	IQ_stMeldung.bMeldFBError_ErrorDiag	:= FALSE;
	IQ_stMeldung.bMeldFBError_ErrorState:= FALSE;
	IQ_stMeldung.sMeldFBError_ErrorDiag	:= '';
	IQ_stMeldung.sMeldFBError_ErrorState:= '';
	
	sFB				:= CONCAT('TwinSAFE Gruppe',INT_TO_STRING(I_nGrpId));
	sFB				:= CONCAT(sFB,' => ');
	sFB				:= CONCAT(sFB,'FB');
	sFB				:= CONCAT(sFB,INT_TO_STRING(I_nFBId));
	sFB				:= CONCAT(sFB,' ');
	sFB				:= CONCAT(sFB,I_sFBName);
	sFB				:= CONCAT(sFB,' => ');

	(* ========================================================= *)
	(* State *)
	CASE I_stInfoData.nMapState OF
		0:	IQ_stMeldung.sMeldFBError_ErrorState	:= 'undefiniert';
			act_State();

		1:	IQ_stMeldung.sMeldFBError_ErrorState	:= 'Run';

		2:	IQ_stMeldung.sMeldFBError_ErrorState	:= 'Stop';

		3:	IQ_stMeldung.sMeldFBError_ErrorState	:= 'Safe';

	ELSE	IQ_stMeldung.sMeldFBError_ErrorState	:= 'Error';
			act_State();
	END_CASE

	(* ========================================================= *)
	(* Diagnose *)
	(*	stInfoData.uiMapDiag	immer gleich 0*)
	CASE I_stInfoData.nMapState OF
		0:	;
	END_CASE

	(* ========================================================= *)
	(*BE*)
END_ACTION

ACTION actInfoConnectionShutDown:
	(* TwinSAFE-Funktionsbaustein FB Connection Shutdown *)
	(* ========================================================= *)

	IQ_stMeldung.bMeldFBError_ErrorDiag	:= FALSE;
	IQ_stMeldung.bMeldFBError_ErrorState:= FALSE;
	IQ_stMeldung.sMeldFBError_ErrorDiag	:= '';
	IQ_stMeldung.sMeldFBError_ErrorState:= '';
	
	sFB				:= CONCAT('TwinSAFE Gruppe',INT_TO_STRING(I_nGrpId));
	sFB				:= CONCAT(sFB,' => ');
	sFB				:= CONCAT(sFB,'FB');
	sFB				:= CONCAT(sFB,INT_TO_STRING(I_nFBId));
	sFB				:= CONCAT(sFB,' ');
	sFB				:= CONCAT(sFB,I_sFBName);
	sFB				:= CONCAT(sFB,' => ');

	(* ========================================================= *)
	(* State *)
	CASE I_stInfoData.nMapState OF
		0:	IQ_stMeldung.sMeldFBError_ErrorState	:= 'undefiniert';
			act_State();

		2:	IQ_stMeldung.sMeldFBError_ErrorState	:= 'Stop';

		3:	IQ_stMeldung.sMeldFBError_ErrorState	:= 'Safe';

		4:	IQ_stMeldung.sMeldFBError_ErrorState	:= 'Error';
			act_State();

		5:	IQ_stMeldung.sMeldFBError_ErrorState	:= 'Reset';

		10:IQ_stMeldung.sMeldFBError_ErrorState	:= 'Active';

		11:IQ_stMeldung.sMeldFBError_ErrorState	:= 'Deactive';

	ELSE	IQ_stMeldung.sMeldFBError_ErrorState	:= 'Error';
			act_State();
	END_CASE

	(* ========================================================= *)
	(* Diagnose *)
	(*	stInfoData.uiMapDiag	immer gleich 0*)
	CASE I_stInfoData.nMapDiag OF
		0: IQ_stMeldung.sMeldFBError_ErrorDiag	 :='-';
	ELSE
		IF I_stInfoData.nMapDiag.0 THEN
			IQ_stMeldung.sMeldFBError_ErrorDiag	:='Diskrepanz Fehler Eingangsgruppe 1 => Safety Input => ';
			IQ_stMeldung.sMeldFBError_ErrorDiag	:= CONCAT(IQ_stMeldung.sMeldFBError_ErrorDiag,I_sNameEinGruppe1);
			act_Diag();
		END_IF
	END_CASE

	(* ========================================================= *)
	(*BE*)
END_ACTION

ACTION actInfoDecoupler:
	(* TwinSAFE-Funktionsbaustein FB Decouple*)
	(* ========================================================= *)

	IQ_stMeldung.bMeldFBError_ErrorDiag	:= FALSE;
	IQ_stMeldung.bMeldFBError_ErrorState:= FALSE;
	IQ_stMeldung.sMeldFBError_ErrorDiag	:= '';
	IQ_stMeldung.sMeldFBError_ErrorState:= '';
	
	sFB				:= CONCAT('TwinSAFE Gruppe',INT_TO_STRING(I_nGrpId));
	sFB				:= CONCAT(sFB,' => ');
	sFB				:= CONCAT(sFB,'FB');
	sFB				:= CONCAT(sFB,INT_TO_STRING(I_nFBId));
	sFB				:= CONCAT(sFB,' ');
	sFB				:= CONCAT(sFB,I_sFBName);
	sFB				:= CONCAT(sFB,' => ');

	(* ========================================================= *)
	(* State *)
	CASE I_stInfoData.nMapState OF
		0:	IQ_stMeldung.sMeldFBError_ErrorState	:= 'undefiniert';
			act_State();

		1:	IQ_stMeldung.sMeldFBError_ErrorState	:= 'Run';

		2:	IQ_stMeldung.sMeldFBError_ErrorState	:= 'Stop';

	ELSE	IQ_stMeldung.sMeldFBError_ErrorState	:= 'Error';
			act_State();
	END_CASE

	(* ========================================================= *)
	(* Diagnose *)
	(*	stInfoData.uiMapDiag	immer gleich 0*)
	CASE I_stInfoData.nMapState OF
		0:	;
	END_CASE

	(* ========================================================= *)
	(*BE*)
END_ACTION

ACTION actInfoEDM:
	(* TwinSAFE-Funktionsbaustein FB EDM *)
	(* ========================================================= *)

	IQ_stMeldung.bMeldFBError_ErrorDiag	:= FALSE;
	IQ_stMeldung.bMeldFBError_ErrorState:= FALSE;
	IQ_stMeldung.sMeldFBError_ErrorDiag	:= '';
	IQ_stMeldung.sMeldFBError_ErrorState:= '';

	sFB				:= CONCAT('TwinSAFE Gruppe',INT_TO_STRING(I_nGrpId));
	sFB				:= CONCAT(sFB,' => ');
	sFB				:= CONCAT(sFB,'FB');
	sFB				:= CONCAT(sFB,INT_TO_STRING(I_nFBId));
	sFB				:= CONCAT(sFB,' ');
	sFB				:= CONCAT(sFB,I_sFBName);
	sFB				:= CONCAT(sFB,' => ');

	(* ========================================================= *)
	(* State *)
	CASE I_stInfoData.nMapState OF
		0:	IQ_stMeldung.sMeldFBError_ErrorState	:= 'undefiniert';
			act_State();

		2:	IQ_stMeldung.sMeldFBError_ErrorState	:= 'Stop';

		4:	IQ_stMeldung.sMeldFBError_ErrorState	:= 'Error';
			act_State();

		5:	IQ_stMeldung.sMeldFBError_ErrorState	:= 'Reset';

		14:IQ_stMeldung.sMeldFBError_ErrorState	:= 'MON_OFF';

		15:IQ_stMeldung.sMeldFBError_ErrorState	:= 'MON_ON';

	ELSE	IQ_stMeldung.sMeldFBError_ErrorState	:= 'Error';
			act_State();
	END_CASE

	(* ========================================================= *)
	(* Diagnose *)
	CASE I_stInfoData.nMapDiag OF
		0: ;
	ELSE
		IF I_stInfoData.nMapDiag.0 THEN
			IQ_stMeldung.sMeldFBError_ErrorDiag	:='Switch OFF Timer abgelaufen';
			act_Diag();
		END_IF
		IF I_stInfoData.nMapDiag.1 THEN
			IQ_stMeldung.sMeldFBError_ErrorDiag	:='Switch ON Timer abgelaufen';
			act_Diag();
		END_IF
	END_CASE

	(* ========================================================= *)
	(*BE*)
END_ACTION

ACTION actInfoEStop:
	(* TwinSAFE-Funktionsbaustein FB EStop *)
	(* ========================================================= *)

	IQ_stMeldung.bMeldFBError_ErrorDiag	:= FALSE;
	IQ_stMeldung.bMeldFBError_ErrorState:= FALSE;
	IQ_stMeldung.sMeldFBError_ErrorDiag	:= '';
	IQ_stMeldung.sMeldFBError_ErrorState:= '';

	sFB				:= CONCAT('TwinSAFE Gruppe',INT_TO_STRING(I_nGrpId));
	sFB				:= CONCAT(sFB,' => ');
	sFB				:= CONCAT(sFB,'FB');
	sFB				:= CONCAT(sFB,INT_TO_STRING(I_nFBId));
	sFB				:= CONCAT(sFB,' ');
	sFB				:= CONCAT(sFB,I_sFBName);
	sFB				:= CONCAT(sFB,' => ');
	(* ========================================================= *)
	(* State *)
	CASE I_stInfoData.nMapState OF
		0:	IQ_stMeldung.sMeldFBError_ErrorState	:= 'undefiniert';
			act_State();

		1:	IQ_stMeldung.sMeldFBError_ErrorState	:= 'Run';

		2:	IQ_stMeldung.sMeldFBError_ErrorState	:= 'Stop';

		3:	IQ_stMeldung.sMeldFBError_ErrorState	:= 'Safe';

		4:	IQ_stMeldung.sMeldFBError_ErrorState	:= 'Error';
			act_State();

		5:	IQ_stMeldung.sMeldFBError_ErrorState	:= 'Reset';

		6:	IQ_stMeldung.sMeldFBError_ErrorState	:= 'Start';

		8:	IQ_stMeldung.sMeldFBError_ErrorState	:= 'DelayOut';

	ELSE	IQ_stMeldung.sMeldFBError_ErrorState	:= 'Error';
			act_State();
	END_CASE

	(* ========================================================= *)
	(* Diagnose *)
	CASE I_stInfoData.nMapDiag OF
		0: IQ_stMeldung.sMeldFBError_ErrorDiag :='-';
	ELSE
		IF I_stInfoData.nMapDiag.0 THEN
			IQ_stMeldung.sMeldFBError_ErrorDiag	:='Diskrepanz Fehler Eingangsgruppe 1 => Safety Input => ';
			IQ_stMeldung.sMeldFBError_ErrorDiag	:= CONCAT(IQ_stMeldung.sMeldFBError_ErrorDiag,I_sNameEinGruppe1);
			act_Diag();
		END_IF

		IF I_stInfoData.nMapDiag.1 THEN
			IQ_stMeldung.sMeldFBError_ErrorDiag	:='Diskrepanz Fehler Eingangsgruppe 2 => Safety Input => ';
			IQ_stMeldung.sMeldFBError_ErrorDiag	:= CONCAT(IQ_stMeldung.sMeldFBError_ErrorDiag,I_sNameEinGruppe2);
			act_Diag();
		END_IF

		IF I_stInfoData.nMapDiag.2 THEN
			IQ_stMeldung.sMeldFBError_ErrorDiag	:='Diskrepanz Fehler Eingangsgruppe 3 => Safety Input => ';
			IQ_stMeldung.sMeldFBError_ErrorDiag	:= CONCAT(IQ_stMeldung.sMeldFBError_ErrorDiag,I_sNameEinGruppe3);
			act_Diag();
		END_IF

		IF I_stInfoData.nMapDiag.3 THEN
			IQ_stMeldung.sMeldFBError_ErrorDiag	:='Diskrepanz Fehler Eingangsgruppe 4 => Safety Input => ';
			IQ_stMeldung.sMeldFBError_ErrorDiag	:= CONCAT(IQ_stMeldung.sMeldFBError_ErrorDiag,I_sNameEinGruppe4);
			act_Diag();
		END_IF

		IF I_stInfoData.nMapDiag.4 THEN
			IQ_stMeldung.sMeldFBError_ErrorDiag	:='Rueckfuehrkreis Fehler EDM1 => Safety Input => ';
			IQ_stMeldung.sMeldFBError_ErrorDiag	:= CONCAT(IQ_stMeldung.sMeldFBError_ErrorDiag,I_sNameEMD1);
			act_Diag();
		END_IF

		IF I_stInfoData.nMapDiag.5 THEN
			IQ_stMeldung.sMeldFBError_ErrorDiag	:='Rueckfuehrkreis Fehler EDM2 => Safety Input => ';
			IQ_stMeldung.sMeldFBError_ErrorDiag	:= CONCAT(IQ_stMeldung.sMeldFBError_ErrorDiag,I_sNameEMD2);
			act_Diag();
		END_IF
	END_CASE

	(* ========================================================= *)
	(*BE*)
END_ACTION

ACTION actInfoMON:
	(* TwinSAFE-Funktionsbaustein FB MOM *)
	(* ========================================================= *)

	IQ_stMeldung.bMeldFBError_ErrorDiag	:= FALSE;
	IQ_stMeldung.bMeldFBError_ErrorState:= FALSE;
	IQ_stMeldung.sMeldFBError_ErrorDiag	:= '';
	IQ_stMeldung.sMeldFBError_ErrorState:= '';

	sFB				:= CONCAT('TwinSAFE Gruppe',INT_TO_STRING(I_nGrpId));
	sFB				:= CONCAT(sFB,' => ');
	sFB				:= CONCAT(sFB,'FB');
	sFB				:= CONCAT(sFB,INT_TO_STRING(I_nFBId));
	sFB				:= CONCAT(sFB,' ');
	sFB				:= CONCAT(sFB,I_sFBName);
	sFB				:= CONCAT(sFB,' => ');

	(* ========================================================= *)
	(* State *)
	CASE I_stInfoData.nMapState OF
		0:	IQ_stMeldung.sMeldFBError_ErrorState	:= 'undefiniert';
			act_State();

		1:	IQ_stMeldung.sMeldFBError_ErrorState	:= 'Run';

		2:	IQ_stMeldung.sMeldFBError_ErrorState	:= 'Stop';

		3:	IQ_stMeldung.sMeldFBError_ErrorState	:= 'Safe';

		4:	IQ_stMeldung.sMeldFBError_ErrorState	:= 'Error';
			act_State();

		5:	IQ_stMeldung.sMeldFBError_ErrorState	:= 'Reset';

		6:	IQ_stMeldung.sMeldFBError_ErrorState	:= 'Start';

		7:	IQ_stMeldung.sMeldFBError_ErrorState	:= 'ErrorDelay';
			act_State();

		8:	IQ_stMeldung.sMeldFBError_ErrorState	:= 'DelayOut';

		9:	IQ_stMeldung.sMeldFBError_ErrorState	:= 'FuncTest';

	ELSE	IQ_stMeldung.sMeldFBError_ErrorState	:= 'Error';
			act_State();
	END_CASE

	(* ========================================================= *)
	(* Diagnose *)
	CASE I_stInfoData.nMapDiag OF
		0: ;
	ELSE
		IF I_stInfoData.nMapDiag.0 THEN
			IQ_stMeldung.sMeldFBError_ErrorDiag	:='Diskrepanz Fehler Eingangsgruppe 1 => Safety Input => ';
			IQ_stMeldung.sMeldFBError_ErrorDiag	:= CONCAT(IQ_stMeldung.sMeldFBError_ErrorDiag,I_sNameEinGruppe1);
			act_Diag();
		END_IF

		IF I_stInfoData.nMapDiag.1 THEN
			IQ_stMeldung.sMeldFBError_ErrorDiag	:='Diskrepanz Fehler Eingangsgruppe 2 => Safety Input => ';
			IQ_stMeldung.sMeldFBError_ErrorDiag	:= CONCAT(IQ_stMeldung.sMeldFBError_ErrorDiag,I_sNameEinGruppe2);
			act_Diag();
		END_IF

		IF I_stInfoData.nMapDiag.2 THEN
			IQ_stMeldung.sMeldFBError_ErrorDiag	:='Diskrepanz Fehler Secure-Eingangsgruppe => Safety Input => ';
			IQ_stMeldung.sMeldFBError_ErrorDiag	:= CONCAT(IQ_stMeldung.sMeldFBError_ErrorDiag,I_sNameSecGruppe);
			act_Diag();
		END_IF

		IF I_stInfoData.nMapDiag.4 THEN
			IQ_stMeldung.sMeldFBError_ErrorDiag	:='Rueckfuehrkreis Fehler EDM1 => Safety Input => ';
			IQ_stMeldung.sMeldFBError_ErrorDiag	:= CONCAT(IQ_stMeldung.sMeldFBError_ErrorDiag,I_sNameEMD1);
			act_Diag();
		END_IF

		IF I_stInfoData.nMapDiag.5 THEN
			IQ_stMeldung.sMeldFBError_ErrorDiag	:='Rueckfuehrkreis Fehler EDM2 => Safety Input => ';
			IQ_stMeldung.sMeldFBError_ErrorDiag	:= CONCAT(IQ_stMeldung.sMeldFBError_ErrorDiag,I_sNameEMD2);
			act_Diag();
		END_IF
	END_CASE

	(* ========================================================= *)
	(*BE*)
END_ACTION

ACTION actInfoMuting:
	(* TwinSAFE-Funktionsbaustein FB MUTING*)
	(* ========================================================= *)

	IQ_stMeldung.bMeldFBError_ErrorDiag	:= FALSE;
	IQ_stMeldung.bMeldFBError_ErrorState:= FALSE;
	IQ_stMeldung.sMeldFBError_ErrorDiag	:= '';
	IQ_stMeldung.sMeldFBError_ErrorState:= '';

	sFB				:= CONCAT('TwinSAFE Gruppe',INT_TO_STRING(I_nGrpId));
	sFB				:= CONCAT(sFB,' => ');
	sFB				:= CONCAT(sFB,'FB');
	sFB				:= CONCAT(sFB,INT_TO_STRING(I_nFBId));
	sFB				:= CONCAT(sFB,' ');
	sFB				:= CONCAT(sFB,I_sFBName);
	sFB				:= CONCAT(sFB,' => ');

	(* ========================================================= *)
	(* State *)
	CASE I_stInfoData.nMapState OF
		0:	IQ_stMeldung.sMeldFBError_ErrorState	:= 'undefiniert';
			act_State();

		1:	IQ_stMeldung.sMeldFBError_ErrorState	:= 'Run';

		2:	IQ_stMeldung.sMeldFBError_ErrorState	:= 'Stop';

		4:	IQ_stMeldung.sMeldFBError_ErrorState	:= 'Safe';

		5:	IQ_stMeldung.sMeldFBError_ErrorState	:= 'Reset';

		6:	IQ_stMeldung.sMeldFBError_ErrorState	:= 'undefiniert';
			act_State();

		7:	IQ_stMeldung.sMeldFBError_ErrorState	:= 'undefiniert';
			act_State();

		8:	IQ_stMeldung.sMeldFBError_ErrorState	:= 'DelayOut';

		9:	IQ_stMeldung.sMeldFBError_ErrorState	:= 'Muting1';
		10:IQ_stMeldung.sMeldFBError_ErrorState	:= 'Muting2';
		11:IQ_stMeldung.sMeldFBError_ErrorState	:= 'Muting3';
		12:IQ_stMeldung.sMeldFBError_ErrorState	:= 'Muting4';
		13:IQ_stMeldung.sMeldFBError_ErrorState	:= 'Muting5';
		14:IQ_stMeldung.sMeldFBError_ErrorState	:= 'Muting6';
		15:IQ_stMeldung.sMeldFBError_ErrorState	:= 'Muting7';
		16:IQ_stMeldung.sMeldFBError_ErrorState	:= 'Muting8';
		17:IQ_stMeldung.sMeldFBError_ErrorState	:= 'Muting9';

	ELSE 	IQ_stMeldung.sMeldFBError_ErrorState	:= 'Error';
			act_State();
	END_CASE

	(* ========================================================= *)
	(* Diagnose *)
	CASE I_stInfoData.nMapDiag OF
		0: ;
	ELSE
		IF I_stInfoData.nMapDiag.0 THEN
			IQ_stMeldung.sMeldFBError_ErrorDiag	:='Diskrepanz Fehler Muting Eingangsgruppe 1 => Safety Input => ';
			IQ_stMeldung.sMeldFBError_ErrorDiag	:= CONCAT(IQ_stMeldung.sMeldFBError_ErrorDiag,I_sNameEinGruppe1);
			act_Diag();
		END_IF

		IF I_stInfoData.nMapDiag.1 THEN
			IQ_stMeldung.sMeldFBError_ErrorDiag	:='Diskrepanz Fehler OSSD Eingangsgruppe => Safety Input => ';
			IQ_stMeldung.sMeldFBError_ErrorDiag	:= CONCAT(IQ_stMeldung.sMeldFBError_ErrorDiag,I_sNameOSSDEinGruppe);
			act_Diag();
		END_IF

		IF I_stInfoData.nMapDiag.2 THEN
			IQ_stMeldung.sMeldFBError_ErrorDiag	:='Diskrepanz Fehler Muting Eingangsgruppe 2 => Safety Input => ';
			IQ_stMeldung.sMeldFBError_ErrorDiag	:= CONCAT(IQ_stMeldung.sMeldFBError_ErrorDiag,I_sNameEinGruppe2);
			act_Diag();
		END_IF

		IF I_stInfoData.nMapDiag.4 THEN
			IQ_stMeldung.sMeldFBError_ErrorDiag	:='Rueckfuehrkreis Fehler EDM1 => Safety Input => ';
			IQ_stMeldung.sMeldFBError_ErrorDiag	:= CONCAT(IQ_stMeldung.sMeldFBError_ErrorDiag,I_sNameEMD1);
			act_Diag();
		END_IF

		IF I_stInfoData.nMapDiag.5 THEN
			IQ_stMeldung.sMeldFBError_ErrorDiag	:='Rueckfuehrkreis Fehler EDM2 => Safety Input => ';
			IQ_stMeldung.sMeldFBError_ErrorDiag	:= CONCAT(IQ_stMeldung.sMeldFBError_ErrorDiag,I_sNameEMD2);
			act_Diag();
		END_IF

		IF I_stInfoData.nMapDiag.6 THEN
			IQ_stMeldung.sMeldFBError_ErrorDiag	:='Mutingsequenz wurde verletzt';
			act_Diag();
		END_IF

		IF I_stInfoData.nMapDiag.7 THEN
			IQ_stMeldung.sMeldFBError_ErrorDiag	:='Maximale Mutingtime wurde überschritten';
			act_Diag();
		END_IF
	END_CASE

	(* ========================================================= *)
	(*BE*)
END_ACTION

ACTION actInfoOPMode:
	(* TwinSAFE-Funktionsbaustein FB OPMode *)
	(* ========================================================= *)

	IQ_stMeldung.bMeldFBError_ErrorDiag	:= FALSE;
	IQ_stMeldung.bMeldFBError_ErrorState:= FALSE;
	IQ_stMeldung.sMeldFBError_ErrorDiag	:= '';
	IQ_stMeldung.sMeldFBError_ErrorState:= '';

	sFB				:= CONCAT('TwinSAFE Gruppe',INT_TO_STRING(I_nGrpId));
	sFB				:= CONCAT(sFB,' => ');
	sFB				:= CONCAT(sFB,'FB');
	sFB				:= CONCAT(sFB,INT_TO_STRING(I_nFBId));
	sFB				:= CONCAT(sFB,' ');
	sFB				:= CONCAT(sFB,I_sFBName);
	sFB				:= CONCAT(sFB,' => ');

	(* ========================================================= *)
	(* State *)
	CASE I_stInfoData.nMapState OF
		0:	IQ_stMeldung.sMeldFBError_ErrorState	:= 'undefiniert';
			act_State();

		1:	IQ_stMeldung.sMeldFBError_ErrorState	:= 'Run';

		2:	IQ_stMeldung.sMeldFBError_ErrorState	:= 'Stop';

		3:	IQ_stMeldung.sMeldFBError_ErrorState	:= 'Safe';
		
		4:	IQ_stMeldung.sMeldFBError_ErrorState	:= 'ERROR';
			act_State();

		5:	IQ_stMeldung.sMeldFBError_ErrorState	:= 'Reset';

		6:	IQ_stMeldung.sMeldFBError_ErrorState	:= 'Start';

	ELSE	IQ_stMeldung.sMeldFBError_ErrorState	:= 'Error';
			act_State();
	END_CASE

	(* ========================================================= *)
	(* Diagnose *)
	(*	stInfoData.uiMapDiag	immer gleich 0*)
	CASE I_stInfoData.nMapState OF
		0: ;
	ELSE
		IF I_stInfoData.nMapDiag.0 THEN
			IQ_stMeldung.sMeldFBError_ErrorDiag	:= 'Diskrepanzueberwachungsfehler';
			act_Diag();
		END_IF
	END_CASE

	(* ========================================================= *)
	(*BE*)
END_ACTION

ACTION actInfoOR:
	(* TwinSAFE-Funktionsbaustein FB OR *)
	(* ========================================================= *)

	IQ_stMeldung.bMeldFBError_ErrorDiag	:= FALSE;
	IQ_stMeldung.bMeldFBError_ErrorState:= FALSE;
	IQ_stMeldung.sMeldFBError_ErrorDiag	:= '';
	IQ_stMeldung.sMeldFBError_ErrorState:= '';

	sFB				:= CONCAT('TwinSAFE Gruppe',INT_TO_STRING(I_nGrpId));
	sFB				:= CONCAT(sFB,' => ');
	sFB				:= CONCAT(sFB,'FB');
	sFB				:= CONCAT(sFB,INT_TO_STRING(I_nFBId));
	sFB				:= CONCAT(sFB,' ');
	sFB				:= CONCAT(sFB,I_sFBName);
	sFB				:= CONCAT(sFB,' => ');

	(* ========================================================= *)
	(* State *)
	CASE I_stInfoData.nMapState OF
		0:	IQ_stMeldung.sMeldFBError_ErrorState	:= 'undefiniert';
			act_State();

		1:	IQ_stMeldung.sMeldFBError_ErrorState	:= 'Run';

		2:	IQ_stMeldung.sMeldFBError_ErrorState	:= 'Stop';

		3:	IQ_stMeldung.sMeldFBError_ErrorState	:= 'Safe';

	ELSE	IQ_stMeldung.sMeldFBError_ErrorState	:= 'ERROR';
			act_State();
	END_CASE

	(* ========================================================= *)
	(* Diagnose *)
	(*	stInfoData.uiMapDiag	immer gleich 0*)
	CASE I_stInfoData.nMapState OF
		0:	;
	END_CASE

	(* ========================================================= *)
	(*BE*)
END_ACTION

ACTION actInfoRS:
	(* TwinSAFE-Funktionsbaustein FB RS *)
	(* ========================================================= *)

	IQ_stMeldung.bMeldFBError_ErrorDiag	:= FALSE;
	IQ_stMeldung.bMeldFBError_ErrorState:= FALSE;
	IQ_stMeldung.sMeldFBError_ErrorDiag	:= '';
	IQ_stMeldung.sMeldFBError_ErrorState:= '';

	sFB				:= CONCAT('TwinSAFE Gruppe',INT_TO_STRING(I_nGrpId));
	sFB				:= CONCAT(sFB,' => ');
	sFB				:= CONCAT(sFB,'FB');
	sFB				:= CONCAT(sFB,INT_TO_STRING(I_nFBId));
	sFB				:= CONCAT(sFB,' ');
	sFB				:= CONCAT(sFB,I_sFBName);
	sFB				:= CONCAT(sFB,' => ');

	(* ========================================================= *)
	(* State *)
	CASE I_stInfoData.nMapState OF
		0:	IQ_stMeldung.sMeldFBError_ErrorState	:= 'undefiniert';
			act_State();

		2:	IQ_stMeldung.sMeldFBError_ErrorState	:= 'Stop';

		3:	IQ_stMeldung.sMeldFBError_ErrorState	:= 'Safe';

		9:	IQ_stMeldung.sMeldFBError_ErrorState	:= 'Set';

	ELSE	IQ_stMeldung.sMeldFBError_ErrorState	:= 'Error';
			act_State();
	END_CASE

	(* ========================================================= *)
	(* Diagnose *)
	(*	stInfoData.uiMapDiag	immer gleich 0*)
	CASE I_stInfoData.nMapState OF
		0:	;
	END_CASE

	(* ========================================================= *)
	(*BE*)
END_ACTION

ACTION actInfoSR:
	(* TwinSAFE-Funktionsbaustein FB SR *)
	(* ========================================================= *)

	IQ_stMeldung.bMeldFBError_ErrorDiag	:= FALSE;
	IQ_stMeldung.bMeldFBError_ErrorState:= FALSE;
	IQ_stMeldung.sMeldFBError_ErrorDiag	:= '';
	IQ_stMeldung.sMeldFBError_ErrorState:= '';

	sFB				:= CONCAT('TwinSAFE Gruppe',INT_TO_STRING(I_nGrpId));
	sFB				:= CONCAT(sFB,' => ');
	sFB				:= CONCAT(sFB,'FB');
	sFB				:= CONCAT(sFB,INT_TO_STRING(I_nFBId));
	sFB				:= CONCAT(sFB,' ');
	sFB				:= CONCAT(sFB,I_sFBName);
	sFB				:= CONCAT(sFB,' => ');

	(* ========================================================= *)
	(* State *)
	CASE I_stInfoData.nMapState OF
		0:	IQ_stMeldung.sMeldFBError_ErrorState	:= 'undefiniert';
			act_State();

		2:	IQ_stMeldung.sMeldFBError_ErrorState	:= 'Stop';

		3:	IQ_stMeldung.sMeldFBError_ErrorState	:= 'Safe';

		9:	IQ_stMeldung.sMeldFBError_ErrorState	:= 'Set';

	ELSE	IQ_stMeldung.sMeldFBError_ErrorState	:= 'Error';
			act_State();
	END_CASE

	(* ========================================================= *)
	(* Diagnose *)
	(*	stInfoData.uiMapDiag	immer gleich 0*)
	CASE I_stInfoData.nMapState OF
		0:	;
	END_CASE

	(* ========================================================= *)
	(*BE*)
END_ACTION

ACTION actInfoTOF:
	(* TwinSAFE-Funktionsbaustein FB TON *)
	(* ========================================================= *)

	IQ_stMeldung.bMeldFBError_ErrorDiag	:= FALSE;
	IQ_stMeldung.bMeldFBError_ErrorState:= FALSE;
	IQ_stMeldung.sMeldFBError_ErrorDiag	:= '';
	IQ_stMeldung.sMeldFBError_ErrorState:= '';

	sFB				:= CONCAT('TwinSAFE Gruppe',INT_TO_STRING(I_nGrpId));
	sFB				:= CONCAT(sFB,' => ');
	sFB				:= CONCAT(sFB,'FB');
	sFB				:= CONCAT(sFB,INT_TO_STRING(I_nFBId));
	sFB				:= CONCAT(sFB,' ');
	sFB				:= CONCAT(sFB,I_sFBName);
	sFB				:= CONCAT(sFB,' => ');

	(* ========================================================= *)
	(* State *)
	CASE I_stInfoData.nMapState OF
		0:	IQ_stMeldung.sMeldFBError_ErrorState	:= 'undefiniert';
			act_State();

		1:	IQ_stMeldung.sMeldFBError_ErrorState	:= 'Run';

		2:	IQ_stMeldung.sMeldFBError_ErrorState	:= 'Stop';

		3:	IQ_stMeldung.sMeldFBError_ErrorState	:= 'Safe';

		9:	IQ_stMeldung.sMeldFBError_ErrorState	:= 'Delay_Out';

	ELSE	IQ_stMeldung.sMeldFBError_ErrorState	:= 'Error';
			act_State();
	END_CASE

	(* ========================================================= *)
	(* Diagnose *)
	(*	stInfoData.uiMapDiag	immer gleich 0*)
	CASE I_stInfoData.nMapState OF
		0:	;
	END_CASE

	(* ========================================================= *)
	(*BE*)
END_ACTION

ACTION actInfoTON:
	(* TwinSAFE-Funktionsbaustein FB TON *)
	(* ========================================================= *)

	IQ_stMeldung.bMeldFBError_ErrorDiag	:= FALSE;
	IQ_stMeldung.bMeldFBError_ErrorState:= FALSE;
	IQ_stMeldung.sMeldFBError_ErrorDiag	:= '';
	IQ_stMeldung.sMeldFBError_ErrorState:= '';

	sFB				:= CONCAT('TwinSAFE Gruppe',INT_TO_STRING(I_nGrpId));
	sFB				:= CONCAT(sFB,' => ');
	sFB				:= CONCAT(sFB,'FB');
	sFB				:= CONCAT(sFB,INT_TO_STRING(I_nFBId));
	sFB				:= CONCAT(sFB,' ');
	sFB				:= CONCAT(sFB,I_sFBName);
	sFB				:= CONCAT(sFB,' => ');

	(* ========================================================= *)
	(* State *)
	CASE I_stInfoData.nMapState OF
		0:	IQ_stMeldung.sMeldFBError_ErrorState	:= 'undefiniert';
			act_State();

		1:	IQ_stMeldung.sMeldFBError_ErrorState	:= 'Run';

		2:	IQ_stMeldung.sMeldFBError_ErrorState	:= 'Stop';

		3:	IQ_stMeldung.sMeldFBError_ErrorState	:= 'Safe';

		9:	IQ_stMeldung.sMeldFBError_ErrorState	:= 'Delay_In';

	ELSE	IQ_stMeldung.sMeldFBError_ErrorState	:= 'Error';
			act_State();
	END_CASE

	(* ========================================================= *)
	(* Diagnose *)
	(*	stInfoData.uiMapDiag	immer gleich 0*)
	CASE I_stInfoData.nMapState OF
		0:	;
	END_CASE

	(* ========================================================= *)
	(*BE*)
END_ACTION

ACTION actInfoTwoHand:
	(* TwinSAFE-Funktionsbaustein FB AND*)
	(* ========================================================= *)

	IQ_stMeldung.bMeldFBError_ErrorDiag	:= FALSE;
	IQ_stMeldung.bMeldFBError_ErrorState:= FALSE;
	IQ_stMeldung.sMeldFBError_ErrorDiag	:= '';
	IQ_stMeldung.sMeldFBError_ErrorState:= '';

	sFB				:= CONCAT('TwinSAFE Gruppe',INT_TO_STRING(I_nGrpId));
	sFB				:= CONCAT(sFB,' => ');
	sFB				:= CONCAT(sFB,'FB');
	sFB				:= CONCAT(sFB,INT_TO_STRING(I_nFBId));
	sFB				:= CONCAT(sFB,' ');
	sFB				:= CONCAT(sFB,I_sFBName);
	sFB				:= CONCAT(sFB,' => ');

	(* ========================================================= *)
	(* State *)
	CASE I_stInfoData.nMapState OF
		0:	IQ_stMeldung.sMeldFBError_ErrorState	:= 'undefiniert';
			act_State();

		1:	IQ_stMeldung.sMeldFBError_ErrorState	:= 'Run';

		2:	IQ_stMeldung.sMeldFBError_ErrorState	:= 'Stop';

		3:	IQ_stMeldung.sMeldFBError_ErrorState	:= 'Safe';

		4:	IQ_stMeldung.sMeldFBError_ErrorState	:= 'Error';
			act_State();

		5:	IQ_stMeldung.sMeldFBError_ErrorState	:= 'Reset';

		6:	IQ_stMeldung.sMeldFBError_ErrorState	:= 'Start';

		11:IQ_stMeldung.sMeldFBError_ErrorState	:= '1Button';

		12:IQ_stMeldung.sMeldFBError_ErrorState	:= '2Button';

		13:IQ_stMeldung.sMeldFBError_ErrorState	:= 'Release';

	ELSE	IQ_stMeldung.sMeldFBError_ErrorState	:= 'Error';
			act_State();
	END_CASE

	(* ========================================================= *)
	(* Diagnose *)
	CASE I_stInfoData.nMapDiag OF
		0: ;
	ELSE
		IF I_stInfoData.nMapDiag.0 THEN
			IQ_stMeldung.sMeldFBError_ErrorDiag	:='Diskrepanz Fehler Eingangsgruppe 1 => Safety Input => ';
			IQ_stMeldung.sMeldFBError_ErrorDiag	:= CONCAT(IQ_stMeldung.sMeldFBError_ErrorDiag,I_sNameEinGruppe1);
			act_Diag();
		END_IF

		IF I_stInfoData.nMapDiag.1 THEN
			IQ_stMeldung.sMeldFBError_ErrorDiag	:='Diskrepanz Fehler Eingangsgruppe 2 => Safety Input => ';
			IQ_stMeldung.sMeldFBError_ErrorDiag	:= CONCAT(IQ_stMeldung.sMeldFBError_ErrorDiag,I_sNameEinGruppe2);
			act_Diag();
		END_IF

		IF I_stInfoData.nMapDiag.2 THEN
			IQ_stMeldung.sMeldFBError_ErrorDiag	:='Diskrepanz Fehler zwischen den beiden Eingangsgruppe => Safety Input => ';
			IQ_stMeldung.sMeldFBError_ErrorDiag	:= CONCAT(IQ_stMeldung.sMeldFBError_ErrorDiag,I_sNameEinGruppe1);
			IQ_stMeldung.sMeldFBError_ErrorDiag	:= CONCAT(IQ_stMeldung.sMeldFBError_ErrorDiag,'_');
			IQ_stMeldung.sMeldFBError_ErrorDiag	:= CONCAT(IQ_stMeldung.sMeldFBError_ErrorDiag,I_sNameEinGruppe2);
			act_Diag();
		END_IF
	END_CASE

	(* ========================================================= *)
	(*BE*)
END_ACTION

END_FUNCTION_BLOCK

// POUs/DiagSafety/FB_TwinSAFEGroupInfo
(* Version arrHistory: 
Description: Ethercat-Saftey Diagnose für TwinSAFE-Gruppen
Date			| Version	| created under			| Author				| Remark 
---------------------------------------------------------------------------------------- 
12/09/2011	| 1.1.0		| V2.11.0 (Build 1551)	| T.Löhner			| first release
28.02.2023	| 1.2.0		| V3.1.4024.40				| B.Daut				| Adaptiert für Avalon-HMI Meldesystem
*)
FUNCTION_BLOCK FB_TwinSAFEGroupInfo
VAR_IN_OUT
	IQ_stMeldung	: ST_MeldSafetygruppe;
END_VAR
VAR_INPUT
	I_stInfoData	: ST_TwinSAFE_Group_Info;	// TwinSAFE-Verbindung zu den TwinSAFE-Gruppen
	I_nGrpId			: INT;	// TwinSAFE-Gruppe zur Erstellung der Fehlermeldung
	
	I_bMeldungFreigaben	: BOOL;	// TwinSAFE-Gruppe darf überwacht werden. z.B. bFehlerEtherCATAllg
END_VAR
VAR
	sGrp				: STRING;
	sState_old		: Tc2_System.T_MaxString;	// Zum feststellen einer Änderung und damit einhergehenden Neuauslösung der Meldung
	tonStateChange	: TON;	// Zum feststellen einer Änderung und damit einhergehenden Neuauslösung der Meldung
END_VAR

	(* ========================================================= *)
		actInfo();
	(* ========================================================= *)

ACTION act_State:

	IF IQ_stMeldung.sGruppe	<> sState_old
	THEN
		IQ_stMeldung.bMeldAusg	:= FALSE;
	ELSE
		IQ_stMeldung.bMeldAusg	:= I_bMeldungFreigaben;
	END_IF

	tonStateChange(
		IN:= NOT IQ_stMeldung.bMeldAusg,
		PT:=t#500ms);

	IF tonStateChange.Q THEN
		sState_old	:= IQ_stMeldung.sGruppe	;
	END_IF

	IQ_stMeldung.sGruppe			:= CONCAT('Status: ',IQ_stMeldung.sGruppe	);
	IQ_stMeldung.sGruppe			:= CONCAT(sGrp,IQ_stMeldung.sGruppe	);

	(*BE*)
END_ACTION

ACTION actInfo:
	(* TwinSAFE-Group *)
	(* ========================================================= *)
	IQ_stMeldung.bMeldAusg	:= FALSE;
	IQ_stMeldung.sGruppe		:= '';

	sGrp					:= CONCAT('TwinSAFE Gruppe',INT_TO_STRING(I_nGrpId));
	sGrp					:= CONCAT(sGrp,' => ');

(* ========================================================= *)
	(* State *)
	CASE I_stInfoData.nMapState OF
		1: 	IQ_stMeldung.sGruppe	:='Run';

		2: 	IQ_stMeldung.sGruppe	:='Stop';

		3: 	IQ_stMeldung.sGruppe	:='Safe';

		4: 	IQ_stMeldung.sGruppe	:='Error';
				act_State();

		5: 	IQ_stMeldung.sGruppe	:='Reset';

	ELSE		IQ_stMeldung.sGruppe	:='undefiniert';
				act_State();
	END_CASE

	(* ========================================================= *)
END_ACTION

END_FUNCTION_BLOCK

// POUs/DiagSafety/FB_TwinSAFEKlemmeInfo
(*
Beschreibung :	Dieser Baustein liest die Fehler und CoE-Dateien der lokalen Safety-Klemmen aus.
					Dazu wird der komplette EA-Baum nach Safety-Klemmen durchsucht und automatisch gespeichert.
					Die gefundenen Safety-Komponenten werden im Anschluss nacheinander ausgelesen und Fehler ggf. über die Meldestruktur ausgegeben.
					Dieser FB ist für die Verwendung mit der Avalon-HMI geeignet.
Nutzung des Bausteins:
		1. Bibliotheken Tc2_IoFunctions (fuer: IOF_GetBoxNameByAddr) und TC2_EtherCAT (fuer: FB_CoERead) einfügen
		2. Variable "cAnzSafetyKlemmen" in der "AllgemeineParameter"-Liste anpassen
		3. Beim Aufruf des FBs die Ein-und Ausgänge entsprechend der Kommentare unter VAR_INPUT verknüpfen

Version	History
Date				|	Version		|	created under			|	Author			|	Remark 
---------------------------------------------------------------------------------------- 
11/02/2019		|	1.0.0			|	3.1.4022.27 			|	H.Gennet			|	first release
-	-	-	-	-	-	-	-	-	-	-	-	-	-	-	-	-	-	-	-	-	-	-	-	-	-	-	-	-	-	-	-	-	-	-	-	-	-	-	-	-	-	-	-	- 			
21/02/2019		|	1.0.1			|	3.1.4022.28				|	H.Gennet			|	Automatische Formatierung der AMSNetId
																									Input zum Starten des Bausteins (I_bStartInit)
																									Umbenennung Action c_ und f_ (Ergaenzung um EL6910 und AX5806)
																									Umbenennung Ausgangsarray in Q_arrTwinSAFeKlemmenMeldungen
																									nFbMeldeId wird als Input hinzugefuegt -> I_nFbMeldeId
-	-	-	-	-	-	-	-	-	-	-	-	-	-	-	-	-	-	-	-	-	-	-	-	-	-	-	-	-	-	-	-	-	-	-	-	-	-	-	-	-	-	-	-	- 		
17/04/2019		|	1.1.0			|	3.1.4022.29 			|	B.Daut			|	Ergänzung von Q_arrTwinSAFEKlemmenMeldeTexte als Stringarray
																									Q_arrTwinSAFeKlemmenMeldungen als BOOL-Array, machte mehr Sinn
-	-	-	-	-	-	-	-	-	-	-	-	-	-	-	-	-	-	-	-	-	-	-	-	-	-	-	-	-	-	-	-	-	-	-	-	-	-	-	-	-	-	-	-	- 
17/11/2022		|	1.2.0			|	3.1.4024.35 			|	B.Daut			|	neues Meldesystem und neue Klemme EL2912
30/04/2024		|	1.3.0			|	3.1.4024.50				|	B.Daut			|	Diagnosedaten auslesen für alle neueren Safetyklemmen über arbeitet. Ging vorher garnicht. EL1918, EL2911, EL2912, EP2918, EP1918, EP1957, EL6910

*)
FUNCTION_BLOCK FB_TwinSAFEKlemmeInfo
VAR
	(*Timer*)
	tonCoeReadStart 		: Tc2_Standard.TON;		(*Timer für Aktualisierungsrate der Daten*)

	(*Coe-Read*)	
	fbCoeRead     			: Tc2_EtherCAT.FB_EcCoESdoRead;	(*Baustein zum Auslesen der CoE-Daten*)
	nCOEIndex				: WORD ; 	(* Index des Objektes, das gelesen werden soll.*)
	nCoESubIndex			: BYTE ; 	(* Subindex des Objektes, das gelesen werden soll*)
	nCoeReadErrId   		: UDINT;		(*Error ID des CoE-Bausteins*)
	nLastErrIDTemp			: UDINT;		(*letzte Error ID des CoE-Read-Bausteins*)
	bCoeReadError   		: BOOL;		(*Error bei dem CoE-Read-Baustein*)
	nReadBuf         		: UDINT;		(*Puffer des CoE-Read Bausteins*)
	sReadBufString			: Tc2_System.T_MaxString;	(*Puffer des CoE-Read Bausteins als String*)
	nDiagMessage			: BYTE;	// Nummer der aktuellen Diagnosemeldung
	
	nChannelDiag			: WORD;	// Laufvariable für den Kanal, der bearbeitet werden soll
	bModuleFaultActive	: BOOL;	// ModuleFault von einem Kanal ist aktiv.
	arrModuleFault			: ARRAY[1..8] OF BOOL;	// ModuleFault ist aktiv. Klemme hat einen Fehler
	arrModuleFaultLink	: ARRAY[1..8] OF BOOL;	// ModuleFaultLink ist aktiv. Der Kanal kann auch abgeschaltet sein, weil ein anderer Kanal einen Fehler hat
	
	(*IO-Funktion*)
	fbGetSlaveName 		: Tc2_IoFunctions.IOF_GetBoxNameByAddr;
	
	(*Safety-Klemmen*)
	arrSafetyKlemmeInfo	: ARRAY [1..cAnzSafetyKlemmen] OF ST_TwinSAFEKlemmenInfo;	(*Informationen und Fehlerspeicher der einzelnen Klemmen*)

	(*Hilfsvariablen zum Konvertieren der AmsNetId zu T_AmsNetId*)
	sEtherCatNetID			: Tc2_System.T_MaxString;	
	sEtherCatNetIDTeil1	: Tc2_System.T_MaxString;
	sEtherCatNetIDTeil2	: Tc2_System.T_MaxString;
		
	(*Zustandsvariablen*)
	bBusy						: BOOL;	(*Bit wird gesetzt, solange eine Klemme ausgelesen wird*)
	bKlemmenAusgelesen	: BOOL;	(*Gibt Status der Initialisierung an -> Wenn TRUE, dann ist das Initialisieren abgeschlossen*)
	bNeuerFehler			: BOOL;	(*Angabe, ob es bei dem Durchlauf einen neuen Fehler gibt*)
	bSchreiben				: BOOL;	(*Zustandsvariable Uebertragung der Fehler in Ausgangsarray*)
	bCoeReadStart			: BOOL;	(*Verknuepft mit Timer zum Starten Auslesevorgang Fehler Klemme*)
	
	(*Zaehlvariablen*)
	nAktKlemme				: INT	:= 1;	(*Zaehlvariable mit aktueller Klemme*)
	nFehlerIdx				: INT	:= 1;	(*Zaehlvariable fuer die Fehler einer Klemme*)
	nStateDatenAuslesen	: INT;	(*Zählvariable für das Auslesen der CoE-Dateien*)
	nFehlerIndex			: INT	:= 1;	(*Zaehlvariable fuer aktuellen Fehler*)
	nAnzFehlerGesamt		: INT;	(*Zaehlvariable fuer Anzahl aller TwinSAFE Klemmen*)
	nSafetyKlemmeNr		: UINT;	(*Zaehlvariable der aktuell auszulesenden Klemme*)
	nAnzSafetyKlemmen 	: INT	:= 0; 	(*Zaehlvariable Anzahl Safety Klemmen*)
	nSlaveAddr				: UINT; 	(* Feste Adresse des EtherCAT Slaves an den das SDO-Upload Kommando geschickt werden soll.*)(*zB.: 1006*)
	
	(*Zwischenspeicher*)
	sName						: Tc2_System.T_MaxString;	(*Speicher Name der Klemme im System-Manager*)
	sMeldSpeich 			: Tc2_System.T_MaxString;	(*Speicher der Fehlermeldung*)
	nAnzahlAchsen			: INT;				// Anzahl der Achsen bei AX5805
	nAktAchse				: INT;				// Aktuelle Achse zum Fehler-Auslesen AX5805
	
	// Meldungen
	sKlarTextCoeMeldung	: Tc2_System.T_MaxString;
END_VAR
VAR CONSTANT
	cMaxTemperatur			: UDINT := 90;	// Maximale Temperatur - Manuelle Eingabe
END_VAR
VAR_INPUT
	I_nAnzklemmen			: UINT ;				// Verknüpfen mit IO-Device(x)-InfoData-CfgSlaveCount	(z.B. TIID^Device 3 (EtherCAT)^InfoData^CfgSlaveCount)
	I_AmsNetId				: AMSNETID;			// Verknüpfen mit IO-Device(x)-InfoData-AmsNetId			(z.B. TIID^Device 3 (EtherCAT)^InfoData^AmsNetId)
	I_nDeviceID				: UINT;				// Verknüpfen mit IO-Device(x)-InfoData-DevId				(z.B. TIID^Device 3 (EtherCAT)^InfoData^DevId)
	I_timeAktualiserung	: TIME := T#4S;	// Aktualisierungzeit der Daten - Bei hoher Auslastung kann die Zeit erhöht werden
	I_bStartInit			: BOOL;				// Starten der Initialisierung - verknüpfen z.B. mit NOT bEtherCatFehler
END_VAR
VAR_IN_OUT
	IQ_Meldung				: ARRAY [0..cAnzSafetyKlemmen] OF ST_MeldKlemme;	// Meldeausgang kompatibel mit arrMeldKlemmen aus den Avalon-Meldungen
END_VAR


a_Initialisierung();

b_Ablauf();

ACTION a_Initialisierung:
(*AmsNetId Auslesen - Formatierung vom Typ AmsNetId zu T_AmsNetId*)
sEtherCatNetID := F_CreateAmsNetId(I_AmsNetId);
	
(*Suchen der einzelnen Safety-Klemmen*)	
IF NOT bKlemmenAusgelesen 
	AND I_bStartInit THEN
		IF nSafetyKlemmeNr < (I_nAnzKlemmen -1) THEN
			nSlaveAddr		:= 1002 + nSafetyKlemmeNr;	(*Die Slave-Adresse wird von 1002 ausgehend durchgezählt (1000 = Device, 1001 = Koppler*)	
		
			nCoeIndex		:= 16#1008;	//Index fuer die Bezeichnung der Klemme
			nCoESubIndex	:= 16#0;	// Subindex Klemmenbezeichnung
			
			// Auslesen des Typs. EL1904, EL2904 usw...
			fbCoeRead(
				sNetId		:= sEtherCatNetID,
				nSlaveAddr 	:= nSlaveAddr,
				nIndex		:= nCoEIndex,
				nSubIndex 	:= nCoESubIndex,
				pDstBuf		:= ADR(sReadBufString),
				cbBufLen		:= SIZEOF(sReadBufString),
				bExecute		:= TRUE,
		   	
				bError		=> bCoeReadError,
				nErrId		=> nCoeReadErrId
			);
			
			fbCoeRead(bExecute:= FALSE);	
			
			fbGetSlaveName(
				NETID		:= '',
				DEVICEID	:= I_nDeviceID,
				BOXADDR	:= nSlaveAddr,
				START		:= TRUE,
				TMOUT		:= T#1S,		
				BOXNAME	=> sName
		  );
			
				 
			IF NOT fbCoeRead.bBusy 
				AND NOT fbGetSlaveName.BUSY THEN		(* Bausteine sind durchgelaufen *)
				IF fbCoeRead.bError THEN				(* Wenn ein Error vorliegt, wird dieser ausgegeben - Ein Error tritt auch auf, wenn Klemmen ohne CoE-Daten ausgelesen werden *)
					nLastErrIDTemp 						(* Zwischenspeichern der Error ID des CoE-Read Bausteins*)
						:= fbCoeRead.nErrID;
					bCoeReadError := TRUE;
				ELSE
					bCoeReadError := FALSE;
				// Abfrage des Buffers auf die ausgelesene Klemmenbezeichnung
					IF LEFT(sReadBufString,6) = 'EL6900' THEN
						nAnzSafetyKlemmen := nAnzSafetyKlemmen + 1;
						arrSafetyKlemmeInfo[nAnzSafetyKlemmen].nAdresse := nSlaveAddr; (*Adresse und Klemmentyp werden gespeichert*)
						arrSafetyKlemmeInfo[nAnzSafetyKlemmen].eTyp := E_SafetyType.eEL6900;
						arrSafetyKlemmeInfo[nAnzSafetyKlemmen].sName := fbGetSlaveName.BOXNAME;
					ELSIF LEFT(sReadBufString,6) = 'EL6910' THEN
						nAnzSafetyKlemmen := nAnzSafetyKlemmen + 1;
						arrSafetyKlemmeInfo[nAnzSafetyKlemmen].nAdresse := nSlaveAddr;	(*Adresse und Klemmentyp werden gespeichert*)
						arrSafetyKlemmeInfo[nAnzSafetyKlemmen].eTyp := E_SafetyType.eEL6910;
						arrSafetyKlemmeInfo[nAnzSafetyKlemmen].sName := fbGetSlaveName.BOXNAME;
					ELSIF LEFT(sReadBufString,6) = 'EL1904' THEN
						nAnzSafetyKlemmen := nAnzSafetyKlemmen + 1;
						arrSafetyKlemmeInfo[nAnzSafetyKlemmen].nAdresse := nSlaveAddr;	(*Adresse und Klemmentyp werden gespeichert*)
						arrSafetyKlemmeInfo[nAnzSafetyKlemmen].eTyp := E_SafetyType.eEL1904;
						arrSafetyKlemmeInfo[nAnzSafetyKlemmen].sName := fbGetSlaveName.BOXNAME;
					ELSIF LEFT(sReadBufString,6) = 'EL2904' THEN
						nAnzSafetyKlemmen := nAnzSafetyKlemmen + 1;
						arrSafetyKlemmeInfo[nAnzSafetyKlemmen].nAdresse := nSlaveAddr;	(*Adresse und Klemmentyp werden gespeichert*)
						arrSafetyKlemmeInfo[nAnzSafetyKlemmen].eTyp := E_SafetyType.eEL2904;
						arrSafetyKlemmeInfo[nAnzSafetyKlemmen].sName := fbGetSlaveName.BOXNAME;
					ELSIF LEFT(sReadBufString,6) = 'EL2911' THEN
						nAnzSafetyKlemmen := nAnzSafetyKlemmen + 1;
						arrSafetyKlemmeInfo[nAnzSafetyKlemmen].nAdresse := nSlaveAddr;	(*Adresse und Klemmentyp werden gespeichert*)
						arrSafetyKlemmeInfo[nAnzSafetyKlemmen].eTyp := E_SafetyType.eEL2911;
						arrSafetyKlemmeInfo[nAnzSafetyKlemmen].sName := fbGetSlaveName.BOXNAME;
					ELSIF LEFT(sReadBufString,6) = 'EL2912' THEN
						nAnzSafetyKlemmen := nAnzSafetyKlemmen + 1;
						arrSafetyKlemmeInfo[nAnzSafetyKlemmen].nAdresse := nSlaveAddr;	(*Adresse und Klemmentyp werden gespeichert*)
						arrSafetyKlemmeInfo[nAnzSafetyKlemmen].eTyp := E_SafetyType.eEL2912;
						arrSafetyKlemmeInfo[nAnzSafetyKlemmen].sName := fbGetSlaveName.BOXNAME;
					ELSIF LEFT(sReadBufString,6) = 'AX5805' THEN
						nAnzSafetyKlemmen := nAnzSafetyKlemmen + 1;
						arrSafetyKlemmeInfo[nAnzSafetyKlemmen].nAdresse := nSlaveAddr;	(*Adresse und Klemmentyp werden gespeichert*)
						arrSafetyKlemmeInfo[nAnzSafetyKlemmen].eTyp := 4;
						arrSafetyKlemmeInfo[nAnzSafetyKlemmen].sName := fbGetSlaveName.BOXNAME;
					ELSIF LEFT(sReadBufString,6) = 'AX5806' THEN
						nAnzSafetyKlemmen := nAnzSafetyKlemmen + 1;
						arrSafetyKlemmeInfo[nAnzSafetyKlemmen].nAdresse := nSlaveAddr;	(*Adresse und Klemmentyp werden gespeichert*)
						arrSafetyKlemmeInfo[nAnzSafetyKlemmen].eTyp := E_SafetyType.eAX5806;
						arrSafetyKlemmeInfo[nAnzSafetyKlemmen].sName := fbGetSlaveName.BOXNAME;
					ELSIF LEFT(sReadBufString,6) = 'EL1918' THEN
						nAnzSafetyKlemmen := nAnzSafetyKlemmen + 1;
						arrSafetyKlemmeInfo[nAnzSafetyKlemmen].nAdresse := nSlaveAddr;	(*Adresse und Klemmentyp werden gespeichert*)
						arrSafetyKlemmeInfo[nAnzSafetyKlemmen].eTyp := E_SafetyType.eEL1918;
						arrSafetyKlemmeInfo[nAnzSafetyKlemmen].sName := fbGetSlaveName.BOXNAME;
					ELSIF LEFT(sReadBufString,6) = 'EK1914' THEN
						nAnzSafetyKlemmen := nAnzSafetyKlemmen + 1;
						arrSafetyKlemmeInfo[nAnzSafetyKlemmen].nAdresse := nSlaveAddr;	(*Adresse und Klemmentyp werden gespeichert*)
						arrSafetyKlemmeInfo[nAnzSafetyKlemmen].eTyp := E_SafetyType.eEK1914;
						arrSafetyKlemmeInfo[nAnzSafetyKlemmen].sName := fbGetSlaveName.BOXNAME;
					ELSIF LEFT(sReadBufString,6) = 'EP1908' THEN
						nAnzSafetyKlemmen := nAnzSafetyKlemmen + 1;
						arrSafetyKlemmeInfo[nAnzSafetyKlemmen].nAdresse := nSlaveAddr;	(*Adresse und Klemmentyp werden gespeichert*)
						arrSafetyKlemmeInfo[nAnzSafetyKlemmen].eTyp := E_SafetyType.eEP1908;
						arrSafetyKlemmeInfo[nAnzSafetyKlemmen].sName := fbGetSlaveName.BOXNAME;
					ELSIF LEFT(sReadBufString,6) = 'EP1918' THEN
						nAnzSafetyKlemmen := nAnzSafetyKlemmen + 1;
						arrSafetyKlemmeInfo[nAnzSafetyKlemmen].nAdresse := nSlaveAddr;	(*Adresse und Klemmentyp werden gespeichert*)
						arrSafetyKlemmeInfo[nAnzSafetyKlemmen].eTyp := E_SafetyType.eEP1918;
						arrSafetyKlemmeInfo[nAnzSafetyKlemmen].sName := fbGetSlaveName.BOXNAME;
					ELSIF LEFT(sReadBufString,6) = 'EP1957' THEN
						nAnzSafetyKlemmen := nAnzSafetyKlemmen + 1;
						arrSafetyKlemmeInfo[nAnzSafetyKlemmen].nAdresse := nSlaveAddr;	(*Adresse und Klemmentyp werden gespeichert*)
						arrSafetyKlemmeInfo[nAnzSafetyKlemmen].eTyp := E_SafetyType.eEP1957;
						arrSafetyKlemmeInfo[nAnzSafetyKlemmen].sName := fbGetSlaveName.BOXNAME;
					ELSIF LEFT(sReadBufString,6) = 'EP2918' THEN
						nAnzSafetyKlemmen := nAnzSafetyKlemmen + 1;
						arrSafetyKlemmeInfo[nAnzSafetyKlemmen].nAdresse := nSlaveAddr;	(*Adresse und Klemmentyp werden gespeichert*)
						arrSafetyKlemmeInfo[nAnzSafetyKlemmen].eTyp := E_SafetyType.eEP2918;
						arrSafetyKlemmeInfo[nAnzSafetyKlemmen].sName := fbGetSlaveName.BOXNAME;
					END_IF
				END_IF
				fbGetSlaveName(START := FALSE);
				nSafetyKlemmeNr := nSafetyKlemmeNr + 1;
			END_IF	
		ELSE
			bKlemmenAusgelesen := TRUE; (*Alle Klemmen ausgelesen - Init-Vorgang abgeschlossen*)
		END_IF
END_IF
END_ACTION

ACTION b_Ablauf:
(*Timer fuer Aktualisierungszeit des Bausteins*)
tonCoeReadStart(IN:= NOT bCoeReadStart, PT:= I_timeAktualiserung, Q=> , ET=> );

IF NOT bSchreiben
	AND (tonCoeReadStart.Q
		 OR bCoeReadStart)
	AND bKlemmenAusgelesen
THEN
	bCoeReadStart := TRUE;	// Variable zur Selbsthaltung wird nach Init-Vorgang gesetzt
	
	IF nAktKlemme <= nAnzSafetyKlemmen
		AND nAnzSafetyKlemmen <= cAnzSafetyKlemmen
	THEN
		(*Typ der Klemme auslesen und zugehöriges Programm aufrufen. Parameter muessen nicht uebergeben werden*)
		CASE arrSafetyKlemmeInfo[nAktKlemme].eTyp OF
		E_SafetyType.eEL6900: c_EL6900();
		E_SafetyType.eEL6910: c_EL6910();
		E_SafetyType.eEL1904: d_EL1904();
		E_SafetyType.eEL1918: d_EL1918();
		E_SafetyType.eEK1914: d_EK1914();
		E_SafetyType.eEP1908: d_EP1908();
		E_SafetyType.eEP1918: d_EP1918();
		E_SafetyType.eEP1957: d_EP1957();
		E_SafetyType.eEL2904: e_EL2904();
		E_SafetyType.eEL2911: e_EL2911();
		E_SafetyType.eEL2912: e_EL2912();
		E_SafetyType.eEP2918: e_EP2918();
		E_SafetyType.eAX5805: f_AX5805();
		E_SafetyType.eAX5806: f_AX5806();
		ELSE	// zurzeit noch nicht supportete Klemmen
			arrSafetyKlemmeInfo[nAktKlemme].arrFehler[nFehlerIdx] := TRUE;
			arrSafetyKlemmeInfo[nAktKlemme].arrFehlertext[nFehlerIdx] := CONCAT('Folgende Klemme ist noch nicht supportet: ',TO_STRING(arrSafetyKlemmeInfo[nAktKlemme].sName));
		END_CASE
		
		// Eine Klemme ist abgearbeitet, es wird die naechste Klemme genommen
		IF NOT bBusy
			AND nAktKlemme < nAnzSafetyKlemmen
		THEN
			nAktKlemme := nAktKlemme + 1 ;
		// Ist die letzte Klemme erreicht, wird wieder die erste genommen
		ELSIF NOT bBusy
			AND nAktKlemme = nAnzSafetyKlemmen
		THEN
			nAktKlemme := 1;
			bSchreiben := TRUE;
		END_IF
		
	ELSE
		bSchreiben := TRUE;	// mehr Klemmen ausgelesen als Fehlermeldungen konfiguriert
	END_IF
END_IF

// Sind alle Klemmen kontrolliert, wird kontrolliert, ob sich Fehler geändert haben
IF bSchreiben THEN

	// INIT
	bNeuerFehler	:= FALSE;
	FOR nAnzFehlerGesamt	:= 0 TO cAnzSafetyKlemmen
	DO
		IQ_Meldung[nAnzFehlerGesamt].bMeld	:= FALSE;
		IQ_Meldung[nAnzFehlerGesamt].sMeld	:= '';
	END_FOR

	// Auswerten
	IF nAnzSafetyKlemmen <= cAnzSafetyKlemmen
	THEN
		nAnzFehlerGesamt := 1; (*Zaehlvariable fuer das Ausgangs-Meldungsarray zuruecksetzen fuer naechsten Durchgang*)
		FOR nAktKlemme := 1 TO nAnzSafetyKlemmen DO
			FOR nFehlerIndex := 0 TO (arrSafetyKlemmeInfo[nAktKlemme].nAnzFehler) DO
				IF nAnzFehlerGesamt >= cAnzSafetyKlemmen
				THEN EXIT;	// Bei zu vielen Fehlern, Schleife abbrechen
				END_IF
			
				(*Alle anstehenden Fehler werden in ein gemeinsames Array geschrieben*)
				IF arrSafetyKlemmeInfo[nAktKlemme].arrFehlertext[nFehlerIndex] <> '' 
					 AND arrSafetyKlemmeInfo[nAktKlemme].arrFehler[nFehlerIndex]
					 AND IQ_Meldung[nAnzFehlerGesamt].sMeld	<> arrSafetyKlemmeInfo[nAktKlemme].arrFehlertext[nFehlerIndex]
				THEN	// Anstehenden Fehler ins Meldearray eintragen
					IQ_Meldung[nAnzFehlerGesamt].sMeld	:= arrSafetyKlemmeInfo[nAktKlemme].arrFehlertext[nFehlerIndex];	
					nAnzFehlerGesamt := nAnzFehlerGesamt + 1;
					bNeuerFehler := TRUE;
					
				ELSIF (arrSafetyKlemmeInfo[nAktKlemme].arrFehlertext[nFehlerIndex] <> IQ_Meldung[nAnzFehlerGesamt].sMeld
						AND arrSafetyKlemmeInfo[nAktKlemme].arrFehler[nFehlerIndex])
					OR (IQ_Meldung[nAnzFehlerGesamt].sMeld <> ''
						AND NOT arrSafetyKlemmeInfo[nAktKlemme].arrFehler[nFehlerIndex])
				THEN	// Meldung hat sich geändert, oder die Meldung gibt es nicht mehr
					IQ_Meldung[nAnzFehlerGesamt].sMeld	:= arrSafetyKlemmeInfo[nAktKlemme].arrFehlertext[nFehlerIndex];
					bNeuerFehler := TRUE;
					
				ELSIF arrSafetyKlemmeInfo[nAktKlemme].arrFehlertext[nFehlerIndex] <> '' 
					AND IQ_Meldung[nAnzFehlerGesamt].sMeld = arrSafetyKlemmeInfo[nAktKlemme].arrFehlertext[nFehlerIndex]
				THEN	// Gleicher Fehler wie vorher
					nAnzFehlerGesamt := nAnzFehlerGesamt + 1;
					bNeuerFehler := TRUE;
				END_IF
			END_FOR
		END_FOR
	ELSE	// mehr Klemmen gefunden als Meldungen konfiguriert. Dies als einzigel Meldung ausgeben.
		bNeuerFehler := TRUE;
		IQ_Meldung[1].sMeld	:=
			CONCAT('Es wurden mehr Safetyklemmen gefunden als in den Meldungen parameteriert. Bitte anpassen. Gefunden/Parametriert: ',
			CONCAT(TO_STRING(nAnzSafetyKlemmen),
			CONCAT('/',TO_STRING(cAnzSafetyKlemmen))));
	END_IF
	
	// Wenn ein neuer Fehler erkannt wurde, wird das Datenausgangsarray aktualisiert
	IF bNeuerFehler
	THEN	
		FOR nFehlerIndex := 1 TO nAnzFehlerGesamt DO
			IF IQ_Meldung[nFehlerIndex].sMeld <> ''
			THEN
				IQ_Meldung[nFehlerIndex].bMeld := TRUE;
			ELSE
				IQ_Meldung[nFehlerIndex].bMeld := FALSE;
			END_IF
		END_FOR
	END_IF
	
	(*Fehlerarray der Klemmen wird gelöscht, damit es im nächsten Durchgang neu beschrieben werden kann*)
	FOR nAktKlemme := 1 TO nAnzSafetyKlemmen DO
		FOR nFehlerIndex := 0 TO 10 DO
			arrSafetyKlemmeInfo[nAktKlemme].arrFehler[nFehlerIndex] := FALSE;
			arrSafetyKlemmeInfo[nAktKlemme].arrFehlertext[nFehlerIndex] := ''; 
		END_FOR
	END_FOR
	bSchreiben := FALSE;
	bCoeReadStart := FALSE;
	nAktKlemme := 1;	(*Bei dem nächsten Durchlauf der Klemmen wird wieder die erste Klemme genommen.*)
END_IF
END_ACTION

ACTION c_EL6900:
CASE nStateDatenAuslesen OF 
0:(*EL6900*)
	bBusy 			:= TRUE;
	nCoeIndex		:= 16#FA00; (*Index fuer die Diagnose*)
	nCoESubIndex	:= 16#03;	(*Sensortest-Fehler-Ueberpruefung*)
	
	(*Auslesen der Diagnose-Informationen*)
	fbCoeRead(
	sNetId		:= sEtherCatNetID,
	nSlaveAddr 	:= arrSafetyKlemmeInfo[nAktKlemme].nAdresse,
	nIndex		:= nCoEIndex,
	nSubIndex 	:= nCoESubIndex,
	pDstBuf		:= ADR(nReadBuf),
	cbBufLen	:= SIZEOF(nReadBuf),
	bExecute	:= TRUE,

	bError		=> bCoeReadError,
	nErrId		=> nCoeReadErrId
	);

	fbCoeRead(bExecute:= FALSE);
	
	IF NOT fbCoeRead.bBusy THEN					(* Baustein ist durchgelaufen *)
		IF fbCoeRead.bError THEN				(* Wenn ein Error vorliegt, wird dieser ausgegeben *)
			nLastErrIDTemp := fbCoeRead.nErrID;	(* Error-ID des CoE Reads wird gespeichert*)
			bCoeReadError := TRUE;
		ELSE
			(*Auswertung des Buffers aus dem CoE-Read*)
			IF nReadBuf = (5 OR 6 OR 7) THEN		(* Temperaturfehler haben den Index 5, 6 und 7*)
				arrSafetyKlemmeInfo[nAktKlemme].arrFehler[nFehlerIdx] := TRUE;
				arrSafetyKlemmeInfo[nAktKlemme].arrFehlertext[nFehlerIdx] := 
					CONCAT('Temperaturfehler der Klemme mit Adresse: ', 
						arrSafetyKlemmeInfo[nAktKlemme].sName);
				nFehlerIdx := nFehlerIdx + 1;
			ELSIF nReadBuf = (257 OR 258 OR 259 OR 260) THEN	(*Fehler in der Versorgungsspannung haben den Fehler 257 bis 260*)
				arrSafetyKlemmeInfo[nAktKlemme].arrFehler[nFehlerIdx] := TRUE;
				arrSafetyKlemmeInfo[nAktKlemme].arrFehlertext[nFehlerIdx] := 
					CONCAT('Versorgungsfehler der Klemme mit Adresse: ', 
						arrSafetyKlemmeInfo[nAktKlemme].sName);
				nFehlerIdx := nFehlerIdx + 1;
			END_IF
			bCoeReadError := FALSE;
		END_IF
		nStateDatenAuslesen := nStateDatenAuslesen + 1;
	END_IF
	
1:	
	nCoeIndex		:= 16#F100; (*Index fuer die Diagnose*)
	nCoESubIndex	:= 16#01;	(* Safety-Project State: 0 = Offline, 1 = Run, 2 = Stop, 3 = Start, 4 = Restore, 7 = Fault *)
	
	(*Auslesen der Diagnose-Informationen*)
	fbCoeRead(
	sNetId		:= sEtherCatNetID,
	nSlaveAddr 	:= arrSafetyKlemmeInfo[nAktKlemme].nAdresse,
	nIndex		:= nCoEIndex,
	nSubIndex 	:= nCoESubIndex,
	pDstBuf		:= ADR(nReadBuf),
	cbBufLen	:= SIZEOF(nReadBuf),
	bExecute	:= TRUE,

	bError		=> bCoeReadError,
	nErrId		=> nCoeReadErrId
	);

	fbCoeRead(bExecute:= FALSE);
	
	IF NOT fbCoeRead.bBusy THEN					(* Baustein ist durchgelaufen *)
		IF fbCoeRead.bError THEN				(* Wenn ein Error vorliegt, wird dieser ausgegeben *)
			nLastErrIDTemp := fbCoeRead.nErrID;	(* Error-ID des CoE Reads wird gespeichert*)
			bCoeReadError := TRUE;
		ELSE
			(*Auswertung des Buffers aus dem CoE-Read*)
			IF nReadBuf = 0 THEN	
				arrSafetyKlemmeInfo[nAktKlemme].arrFehler[nFehlerIdx] := TRUE;
				arrSafetyKlemmeInfo[nAktKlemme].arrFehlertext[nFehlerIdx] := 
					CONCAT('Safety Projekt Offline! Adresse Logikklemme: ',
						arrSafetyKlemmeInfo[nAktKlemme].sName);
					nFehlerIdx := nFehlerIdx + 1;
			ELSIF nReadBuf = 2 THEN	
				arrSafetyKlemmeInfo[nAktKlemme].arrFehler[nFehlerIdx] := TRUE;
				arrSafetyKlemmeInfo[nAktKlemme].arrFehlertext[nFehlerIdx] := 
					CONCAT('Safety Projekt Gestoppt! Adresse Logikklemme: ',
						arrSafetyKlemmeInfo[nAktKlemme].sName);
				nFehlerIdx := nFehlerIdx + 1;
			ELSIF nReadBuf = 7 THEN	
				arrSafetyKlemmeInfo[nAktKlemme].arrFehler[nFehlerIdx] := TRUE;
				arrSafetyKlemmeInfo[nAktKlemme].arrFehlertext[nFehlerIdx] := 
					CONCAT('Safety Projekt wurde aufgrund eines schwerwiegenden Fehlers beendet! Adresse Logikklemme: ',
						arrSafetyKlemmeInfo[nAktKlemme].sName);
				nFehlerIdx := nFehlerIdx + 1;
			END_IF
			bCoeReadError := FALSE;
		END_IF
		arrSafetyKlemmeInfo[nAktKlemme].nAnzFehler := nFehlerIdx;
		nStateDatenAuslesen := 0;
		nFehlerIdx := 0; 
		bBusy := FALSE;
	END_IF
END_CASE
END_ACTION

ACTION c_EL6910:
CASE nStateDatenAuslesen OF 
0:	// EL6910 mit einem Diagnosearray im CoE 

	nStateDatenAuslesen := 99;	// Hier gibt es keine Diag-Objekte

1:
	bBusy 			:= TRUE;
	nCoeIndex		:= 16#10F3;	// Index für die Klemmendiagnose
	nCoESubIndex	:= 16#02;	// Index der neusten Meldung
	
	(*Auslesen der Diagnose-Informationen*)
	fbCoeRead(
		sNetId		:= sEtherCatNetID,
		nSlaveAddr 	:= arrSafetyKlemmeInfo[nAktKlemme].nAdresse,
		nIndex		:= nCoEIndex,
		nSubIndex 	:= nCoESubIndex,
		pDstBuf		:= ADR(nDiagMessage),
		cbBufLen		:= SIZEOF(nDiagMessage),
		bExecute		:= TRUE,
	
		bError		=> bCoeReadError,
		nErrId		=> nCoeReadErrId
	);

	fbCoeRead(bExecute:= FALSE);
	
	IF NOT fbCoeRead.bBusy
	THEN	// Baustein ist durchgelaufen
		IF fbCoeRead.bError
		THEN	// Wenn ein Error vorliegt, wird dieser ausgegeben
			nLastErrIDTemp := fbCoeRead.nErrID;	// Error-ID des CoE Reads wird gespeichert
			bCoeReadError := TRUE;
		ELSE
			bCoeReadError := FALSE;
		END_IF
		nStateDatenAuslesen := nStateDatenAuslesen + 1;
	END_IF
	
2:	// 
	nCoeIndex		:= 16#10F3;	// Diagnose History
	//nCoESubIndex	:= 16#06;	// Ab SubIndex 06 geht es los mit den Meldungen
	// Der Index, der im Sub 16#02 drin steht, hat schon den Offset von 16#06. Daher direkt auslesen
	nCoESubIndex	:= nDiagMessage;
	
	(*Auslesen der Diagnose-Informationen*)
	fbCoeRead(
		sNetId		:= sEtherCatNetID,
		nSlaveAddr 	:= arrSafetyKlemmeInfo[nAktKlemme].nAdresse,
		nIndex		:= nCoEIndex,
		nSubIndex 	:= nCoESubIndex,
		pDstBuf		:= ADR(sReadBufString),
		cbBufLen	:= SIZEOF(sReadBufString),
		bExecute	:= TRUE,
	
		bError		=> bCoeReadError,
		nErrId		=> nCoeReadErrId
	);

	fbCoeRead(bExecute:= FALSE);
	
	IF NOT fbCoeRead.bBusy
	THEN	// Baustein ist durchgelaufen
		IF fbCoeRead.bError
		THEN	// Wenn ein Error vorliegt, wird dieser ausgegeben
			nLastErrIDTemp	:= fbCoeRead.nErrID;	(* Error-ID des CoE Reads wird gespeichert*)
			bCoeReadError	:= TRUE;
		ELSE
			arrSafetyKlemmeInfo[nAktKlemme].arrFehler[nFehlerIdx] := TRUE;
			arrSafetyKlemmeInfo[nAktKlemme].arrFehlertext[nFehlerIdx] := 
				CONCAT(sReadBufString,
					arrSafetyKlemmeInfo[nAktKlemme].sName);
			nFehlerIdx := nFehlerIdx + 1;
		END_IF
		bCoeReadError := FALSE;
	END_IF

99:	// Diagnose Fertig

	arrSafetyKlemmeInfo[nAktKlemme].nAnzFehler := nFehlerIdx;
	nStateDatenAuslesen := 0;
	nFehlerIdx := 0; 
	bBusy := FALSE;

END_CASE
END_ACTION

ACTION d_EK1914:
CASE nStateDatenAuslesen OF
0:
	bBusy			:= TRUE;	
	
	nCoeIndex		:= 16#FA80; (*Index fuer die Temperatur*)
	nCoESubIndex	:= 16#1;
	
	(*Auslesen der Temperatur*)
	fbCoeRead(
	sNetId		:= sEtherCatNetID,
	nSlaveAddr 	:= arrSafetyKlemmeInfo[nAktKlemme].nAdresse,
	nIndex		:= nCoEIndex,
	nSubIndex 	:= nCoESubIndex,
	pDstBuf		:= ADR(nReadBuf),
	cbBufLen	:= SIZEOF(nReadBuf),
	bExecute	:= TRUE,

	bError		=> bCoeReadError,
	nErrId		=> nCoeReadErrId
	);
		
	fbCoeRead(bExecute:= FALSE);

	IF NOT fbCoeRead.bBusy THEN					(* Baustein ist durchgelaufen *)
		IF fbCoeRead.bError THEN				(* Wenn ein Error vorliegt, wird dieser ausgegeben *)
			nLastErrIDTemp 
				:= fbCoeRead.nErrID;
			bCoeReadError := TRUE;
		ELSE
			(*Auswertung des Buffers aus dem CoE-Read - Vergleich mit Maximaltemperatur*)
			IF nReadBuf > cMaxTemperatur THEN
				arrSafetyKlemmeInfo[nAktKlemme].arrFehler[nFehlerIdx] := TRUE;
				arrSafetyKlemmeInfo[nAktKlemme].arrFehlertext[nFehlerIdx] := 
					CONCAT('TwinSafe: Maximale Temperatur überschritten an Klemme mit der Adresse: ',
					arrSafetyKlemmeInfo[nAktKlemme].sName);
				nFehlerIdx := nFehlerIdx + 1;
			END_IF
			bCoeReadError := FALSE; 
		END_IF
		nStateDatenAuslesen := nStateDatenAuslesen + 1;	
	END_IF
		
1:
(*Sensortest-Fehler-Überprüfung*)
	nCoeIndex		:= 16#800E; (*Index fuer die Diagnose*)
	nCoESubIndex	:= 16#0A;	(*Sensortest-Fehler-Ueberpruefung*)
	
	(*Auslesen der Diagnose-Informationen*)
	fbCoeRead(
	sNetId		:= sEtherCatNetID,
	nSlaveAddr 	:= arrSafetyKlemmeInfo[nAktKlemme].nAdresse,
	nIndex		:= nCoEIndex,
	nSubIndex 	:= nCoESubIndex,
	pDstBuf		:= ADR(nReadBuf),
	cbBufLen	:= SIZEOF(nReadBuf),
	bExecute	:= TRUE,

	bError		=> bCoeReadError,
	nErrId		=> nCoeReadErrId
	);

	fbCoeRead(bExecute:= FALSE);
	
	IF NOT fbCoeRead.bBusy THEN					(* Baustein ist durchgelaufen *)
		IF fbCoeRead.bError THEN				
			nLastErrIDTemp 
				:= fbCoeRead.nErrID;
			bCoeReadError := TRUE;
		ELSE
			(*Auswertung des Buffers aus dem CoE-Read*)
			IF nReadBuf.0 THEN
				arrSafetyKlemmeInfo[nAktKlemme].arrFehler[nFehlerIdx] := TRUE;
				arrSafetyKlemmeInfo[nAktKlemme].arrFehlertext[nFehlerIdx] := 
					CONCAT('Fehler beim Sensortest der Safety-Klemme! (Adresse: ',
					CONCAT(arrSafetyKlemmeInfo[nAktKlemme].sName,(', Eingang 1)')));
				nFehlerIdx := nFehlerIdx + 1;	
			END_IF
			IF nReadBuf.1 THEN
				arrSafetyKlemmeInfo[nAktKlemme].arrFehler[nFehlerIdx] := TRUE;
				arrSafetyKlemmeInfo[nAktKlemme].arrFehlertext[nFehlerIdx] := 
					CONCAT('Fehler beim Sensortest der Safety-Klemme! (Adresse: ',
					CONCAT(arrSafetyKlemmeInfo[nAktKlemme].sName,(', Eingang 2)')));
				nFehlerIdx := nFehlerIdx + 1;	
			END_IF
			IF nReadBuf.2 THEN
				arrSafetyKlemmeInfo[nAktKlemme].arrFehler[nFehlerIdx] := TRUE;
				arrSafetyKlemmeInfo[nAktKlemme].arrFehlertext[nFehlerIdx] := 
					CONCAT('Fehler beim Sensortest der Safety-Klemme! (Adresse: ',
					CONCAT(arrSafetyKlemmeInfo[nAktKlemme].sName,(', Eingang 3)')));
				nFehlerIdx := nFehlerIdx + 1;
			END_IF	
			IF nReadBuf.3 THEN
				arrSafetyKlemmeInfo[nAktKlemme].arrFehler[nFehlerIdx] := TRUE;
				arrSafetyKlemmeInfo[nAktKlemme].arrFehlertext[nFehlerIdx] := 
					CONCAT('Fehler beim Sensortest der Safety-Klemme! (Adresse: ',
					CONCAT(arrSafetyKlemmeInfo[nAktKlemme].sName,(', Eingang 4)')));
				nFehlerIdx := nFehlerIdx + 1;	
			END_IF
			bCoeReadError := FALSE;
		END_IF
			nStateDatenAuslesen := nStateDatenAuslesen + 1;
	END_IF

2:
	
	nCoeIndex		:= 16#800E; (*Index fuer die Diagnose*)
	nCoESubIndex	:= 16#0B;	(*Fehler bei zweikanaliger Auswertung*)
	
	(*Auslesen der Diagnose-Informationen*)
	fbCoeRead(
	sNetId		:= sEtherCatNetID,
	nSlaveAddr 	:= arrSafetyKlemmeInfo[nAktKlemme].nAdresse,
	nIndex		:= nCoEIndex,
	nSubIndex 	:= nCoESubIndex,
	pDstBuf		:= ADR(nReadBuf),
	cbBufLen	:= SIZEOF(nReadBuf),
	bExecute	:= TRUE,

	bError		=> bCoeReadError,
	nErrId		=> nCoeReadErrId
	);

	fbCoeRead(bExecute:= FALSE);
	
	IF NOT fbCoeRead.bBusy THEN					(* Baustein ist durchgelaufen *)
		IF fbCoeRead.bError THEN				(* Wenn ein Error vorliegt, wird dieser ausgegeben *)
			nLastErrIDTemp 
				:= fbCoeRead.nErrID;
			bCoeReadError := TRUE;
		ELSE
			(*Auswertung des Buffers aus dem CoE-Read*)
			IF nReadBuf.0 THEN
				arrSafetyKlemmeInfo[nAktKlemme].arrFehler[nFehlerIdx] := TRUE;
				arrSafetyKlemmeInfo[nAktKlemme].arrFehlertext[nFehlerIdx] := 
					CONCAT('TwinSAFE: Fehler bei zweikanaliger Auswertung an Adresse:',
					arrSafetyKlemmeInfo[nAktKlemme].sName);
				nFehlerIdx := nFehlerIdx + 1;
			END_IF
			bCoeReadError := FALSE;
		END_IF
			nStateDatenAuslesen := nStateDatenAuslesen + 1;
	END_IF

3:
	nCoeIndex		:= 16#800E; (*Index fuer die Diagnose*)
	nCoESubIndex	:= 16#0C;	(*Fehler bei Trittmattenbetriebsart: Eingangspaar uneinig*)
	
	(*Auslesen der Diagnose-Informationen*)
	fbCoeRead(
	sNetId		:= sEtherCatNetID,
	nSlaveAddr 	:= arrSafetyKlemmeInfo[nAktKlemme].nAdresse,
	nIndex		:= nCoEIndex,
	nSubIndex 	:= nCoESubIndex,
	pDstBuf		:= ADR(nReadBuf),
	cbBufLen	:= SIZEOF(nReadBuf),
	bExecute	:= TRUE,

	bError		=> bCoeReadError,
	nErrId		=> nCoeReadErrId
	);

	fbCoeRead(bExecute:= FALSE);
	IF NOT fbCoeRead.bBusy THEN				(* Baustein ist durchgelaufen *)
		IF fbCoeRead.bError THEN				(* Wenn ein Error vorliegt, wird dieser ausgegeben *)
			nLastErrIDTemp 
				:= fbCoeRead.nErrID;
			bCoeReadError := TRUE;
		ELSE
			(*Auswertung des Buffers aus dem CoE-Read*)
			IF nReadBuf.0 THEN
				arrSafetyKlemmeInfo[nAktKlemme].arrFehler[nFehlerIdx] := TRUE;
				arrSafetyKlemmeInfo[nAktKlemme].arrFehlertext[nFehlerIdx] := 
					CONCAT('TwinSAFE: Fehler bei Trittmattenbetriebsart (Eingangspaar uneinig) an Adresse:',
					arrSafetyKlemmeInfo[nAktKlemme].sName);
				nFehlerIdx := nFehlerIdx + 1;
			END_IF
			bCoeReadError := FALSE;
		END_IF
			nStateDatenAuslesen := nStateDatenAuslesen + 1;
	END_IF

4:	
	nCoeIndex		:= 16#800E; (*Index fuer die Diagnose*)
	nCoESubIndex	:= 16#0D;	(*Fehler bei Trittmattenbetriebsart: Fremdeinspeisung*)
	
	(*Auslesen der Diagnose-Informationen*)
	fbCoeRead(
	sNetId		:= sEtherCatNetID,
	nSlaveAddr 	:= arrSafetyKlemmeInfo[nAktKlemme].nAdresse,
	nIndex		:= nCoEIndex,
	nSubIndex 	:= nCoESubIndex,
	pDstBuf		:= ADR(nReadBuf),
	cbBufLen	:= SIZEOF(nReadBuf),
	bExecute	:= TRUE,

	bError		=> bCoeReadError,
	nErrId		=> nCoeReadErrId
	);

	fbCoeRead(bExecute:= FALSE);
	IF NOT fbCoeRead.bBusy THEN					(* Baustein ist durchgelaufen *)
		IF fbCoeRead.bError THEN				(* Wenn ein Error vorliegt, wird dieser ausgegeben *)
			nLastErrIDTemp 
				:= fbCoeRead.nErrID;
			bCoeReadError := TRUE;
		ELSE
			(*Auswertung des Buffers aus dem CoE-Read*)
			IF nReadBuf.0 THEN
				arrSafetyKlemmeInfo[nAktKlemme].arrFehler[nFehlerIdx] := TRUE;
				arrSafetyKlemmeInfo[nAktKlemme].arrFehlertext[nFehlerIdx] := 
					CONCAT('TwinSAFE: Fehler bei Trittmattenbetriebsart (Fremdeinspeisung) an Adresse:',
					arrSafetyKlemmeInfo[nAktKlemme].sName);
				nFehlerIdx := nFehlerIdx + 1;
			END_IF
			bCoeReadError := FALSE;
		END_IF
		nStateDatenAuslesen := 0;	
		arrSafetyKlemmeInfo[nAktKlemme].nAnzFehler := nFehlerIdx;
		nFehlerIdx := 0;
		bBusy := FALSE;	
	END_IF
END_CASE
END_ACTION

ACTION d_EL1904:
CASE nStateDatenAuslesen OF
0:
	bBusy			:= TRUE;	
	
	nCoeIndex		:= 16#FA80; (*Index fuer die Temperatur*)
	nCoESubIndex	:= 16#1;
	
	(*Auslesen der Temperatur*)
	fbCoeRead(
	sNetId		:= sEtherCatNetID,
	nSlaveAddr 	:= arrSafetyKlemmeInfo[nAktKlemme].nAdresse,
	nIndex		:= nCoEIndex,
	nSubIndex 	:= nCoESubIndex,
	pDstBuf		:= ADR(nReadBuf),
	cbBufLen	:= SIZEOF(nReadBuf),
	bExecute	:= TRUE,

	bError		=> bCoeReadError,
	nErrId		=> nCoeReadErrId
	);
		
	fbCoeRead(bExecute:= FALSE);

	IF NOT fbCoeRead.bBusy THEN					(* Baustein ist durchgelaufen *)
		IF fbCoeRead.bError THEN				(* Wenn ein Error vorliegt, wird dieser ausgegeben *)
			nLastErrIDTemp 
				:= fbCoeRead.nErrID;
			bCoeReadError := TRUE;
		ELSE
			(*Auswertung des Buffers aus dem CoE-Read - Vergleich mit Maximaltemperatur*)
			IF nReadBuf > cMaxTemperatur THEN
				arrSafetyKlemmeInfo[nAktKlemme].arrFehler[nFehlerIdx] := TRUE;
				arrSafetyKlemmeInfo[nAktKlemme].arrFehlertext[nFehlerIdx] := 
					CONCAT('TwinSafe: Maximale Temperatur überschritten an Klemme mit der Adresse: ',
					arrSafetyKlemmeInfo[nAktKlemme].sName);
				nFehlerIdx := nFehlerIdx + 1;
			END_IF
			bCoeReadError := FALSE; 
		END_IF
		nStateDatenAuslesen := nStateDatenAuslesen + 1;	
	END_IF

1:
(*Sensortest-Fehler-Überprüfung*)
	nCoeIndex		:= 16#800E; (*Index fuer die Diagnose*)
	nCoESubIndex	:= 16#0A;	(*Sensortest-Fehler-Ueberpruefung*)
	
	(*Auslesen der Diagnose-Informationen*)
	fbCoeRead(
	sNetId		:= sEtherCatNetID,
	nSlaveAddr 	:= arrSafetyKlemmeInfo[nAktKlemme].nAdresse,
	nIndex		:= nCoEIndex,
	nSubIndex 	:= nCoESubIndex,
	pDstBuf		:= ADR(nReadBuf),
	cbBufLen	:= SIZEOF(nReadBuf),
	bExecute	:= TRUE,

	bError		=> bCoeReadError,
	nErrId		=> nCoeReadErrId
	);

	fbCoeRead(bExecute:= FALSE);
	
	IF NOT fbCoeRead.bBusy THEN					(* Baustein ist durchgelaufen *)
		IF fbCoeRead.bError THEN				
			nLastErrIDTemp 
				:= fbCoeRead.nErrID;
			bCoeReadError := TRUE;
		ELSE
			(*Auswertung des Buffers aus dem CoE-Read*)
			IF nReadBuf.0 THEN
				arrSafetyKlemmeInfo[nAktKlemme].arrFehler[nFehlerIdx] := TRUE;
				arrSafetyKlemmeInfo[nAktKlemme].arrFehlertext[nFehlerIdx] := 
					CONCAT('Fehler beim Sensortest der Safety-Klemme! (Adresse: ',
					CONCAT(arrSafetyKlemmeInfo[nAktKlemme].sName,(', Eingang 1)')));
				nFehlerIdx := nFehlerIdx + 1;	
			END_IF
			IF nReadBuf.1 THEN
				arrSafetyKlemmeInfo[nAktKlemme].arrFehler[nFehlerIdx] := TRUE;
				arrSafetyKlemmeInfo[nAktKlemme].arrFehlertext[nFehlerIdx] := 
					CONCAT('Fehler beim Sensortest der Safety-Klemme! (Adresse: ',
					CONCAT(arrSafetyKlemmeInfo[nAktKlemme].sName,(', Eingang 2)')));
				nFehlerIdx := nFehlerIdx + 1;	
			END_IF
			IF nReadBuf.2 THEN
				arrSafetyKlemmeInfo[nAktKlemme].arrFehler[nFehlerIdx] := TRUE;
				arrSafetyKlemmeInfo[nAktKlemme].arrFehlertext[nFehlerIdx] := 
					CONCAT('Fehler beim Sensortest der Safety-Klemme! (Adresse: ',
					CONCAT(arrSafetyKlemmeInfo[nAktKlemme].sName,(', Eingang 3)')));
				nFehlerIdx := nFehlerIdx + 1;
			END_IF	
			IF nReadBuf.3 THEN
				arrSafetyKlemmeInfo[nAktKlemme].arrFehler[nFehlerIdx] := TRUE;
				arrSafetyKlemmeInfo[nAktKlemme].arrFehlertext[nFehlerIdx] := 
					CONCAT('Fehler beim Sensortest der Safety-Klemme! (Adresse: ',
					CONCAT(arrSafetyKlemmeInfo[nAktKlemme].sName,(', Eingang 4)')));
				nFehlerIdx := nFehlerIdx + 1;	
			END_IF
			bCoeReadError := FALSE;
		END_IF
			nStateDatenAuslesen := nStateDatenAuslesen + 1;
	END_IF


2:
	
	nCoeIndex		:= 16#800E; (*Index fuer die Diagnose*)
	nCoESubIndex	:= 16#0B;	(*Fehler bei zweikanaliger Auswertung*)
	
	(*Auslesen der Diagnose-Informationen*)
	fbCoeRead(
	sNetId		:= sEtherCatNetID,
	nSlaveAddr 	:= arrSafetyKlemmeInfo[nAktKlemme].nAdresse,
	nIndex		:= nCoEIndex,
	nSubIndex 	:= nCoESubIndex,
	pDstBuf		:= ADR(nReadBuf),
	cbBufLen	:= SIZEOF(nReadBuf),
	bExecute	:= TRUE,

	bError		=> bCoeReadError,
	nErrId		=> nCoeReadErrId
	);

	fbCoeRead(bExecute:= FALSE);
	
	IF NOT fbCoeRead.bBusy THEN					(* Baustein ist durchgelaufen *)
		IF fbCoeRead.bError THEN				(* Wenn ein Error vorliegt, wird dieser ausgegeben *)
			nLastErrIDTemp 
				:= fbCoeRead.nErrID;
			bCoeReadError := TRUE;
		ELSE
			(*Auswertung des Buffers aus dem CoE-Read*)
			IF nReadBuf.0 THEN
				arrSafetyKlemmeInfo[nAktKlemme].arrFehler[nFehlerIdx] := TRUE;
				arrSafetyKlemmeInfo[nAktKlemme].arrFehlertext[nFehlerIdx] := 
					CONCAT('TwinSAFE: Fehler bei zweikanaliger Auswertung an Adresse:',
					arrSafetyKlemmeInfo[nAktKlemme].sName);
				nFehlerIdx := nFehlerIdx + 1;
			END_IF
			bCoeReadError := FALSE;
		END_IF
			nStateDatenAuslesen := nStateDatenAuslesen + 1;
	END_IF

3:
	nCoeIndex		:= 16#800E; (*Index fuer die Diagnose*)
	nCoESubIndex	:= 16#0C;	(*Fehler bei Trittmattenbetriebsart: Eingangspaar uneinig*)
	
	(*Auslesen der Diagnose-Informationen*)
	fbCoeRead(
	sNetId		:= sEtherCatNetID,
	nSlaveAddr 	:= arrSafetyKlemmeInfo[nAktKlemme].nAdresse,
	nIndex		:= nCoEIndex,
	nSubIndex 	:= nCoESubIndex,
	pDstBuf		:= ADR(nReadBuf),
	cbBufLen	:= SIZEOF(nReadBuf),
	bExecute	:= TRUE,

	bError		=> bCoeReadError,
	nErrId		=> nCoeReadErrId
	);

	fbCoeRead(bExecute:= FALSE);
	IF NOT fbCoeRead.bBusy THEN				(* Baustein ist durchgelaufen *)
		IF fbCoeRead.bError THEN				(* Wenn ein Error vorliegt, wird dieser ausgegeben *)
			nLastErrIDTemp 
				:= fbCoeRead.nErrID;
			bCoeReadError := TRUE;
		ELSE
			(*Auswertung des Buffers aus dem CoE-Read*)
			IF nReadBuf.0 THEN
				arrSafetyKlemmeInfo[nAktKlemme].arrFehler[nFehlerIdx] := TRUE;
				arrSafetyKlemmeInfo[nAktKlemme].arrFehlertext[nFehlerIdx] := 
					CONCAT('TwinSAFE: Fehler bei Trittmattenbetriebsart (Eingangspaar uneinig) an Adresse:',
					arrSafetyKlemmeInfo[nAktKlemme].sName);
				nFehlerIdx := nFehlerIdx + 1;
			END_IF
			bCoeReadError := FALSE;
		END_IF
			nStateDatenAuslesen := nStateDatenAuslesen + 1;
	END_IF

4:	
	nCoeIndex		:= 16#800E; (*Index fuer die Diagnose*)
	nCoESubIndex	:= 16#0D;	(*Fehler bei Trittmattenbetriebsart: Fremdeinspeisung*)
	
	(*Auslesen der Diagnose-Informationen*)
	fbCoeRead(
	sNetId		:= sEtherCatNetID,
	nSlaveAddr 	:= arrSafetyKlemmeInfo[nAktKlemme].nAdresse,
	nIndex		:= nCoEIndex,
	nSubIndex 	:= nCoESubIndex,
	pDstBuf		:= ADR(nReadBuf),
	cbBufLen	:= SIZEOF(nReadBuf),
	bExecute	:= TRUE,

	bError		=> bCoeReadError,
	nErrId		=> nCoeReadErrId
	);

	fbCoeRead(bExecute:= FALSE);
	IF NOT fbCoeRead.bBusy THEN					(* Baustein ist durchgelaufen *)
		IF fbCoeRead.bError THEN				(* Wenn ein Error vorliegt, wird dieser ausgegeben *)
			nLastErrIDTemp 
				:= fbCoeRead.nErrID;
			bCoeReadError := TRUE;
		ELSE
			(*Auswertung des Buffers aus dem CoE-Read*)
			IF nReadBuf.0 THEN
				arrSafetyKlemmeInfo[nAktKlemme].arrFehler[nFehlerIdx] := TRUE;
				arrSafetyKlemmeInfo[nAktKlemme].arrFehlertext[nFehlerIdx] := 
					CONCAT('TwinSAFE: Fehler bei Trittmattenbetriebsart (Fremdeinspeisung) an Adresse:',
					arrSafetyKlemmeInfo[nAktKlemme].sName);
				nFehlerIdx := nFehlerIdx + 1;
			END_IF
			bCoeReadError := FALSE;
		END_IF
		nStateDatenAuslesen := 0;	
		arrSafetyKlemmeInfo[nAktKlemme].nAnzFehler := nFehlerIdx;
		nFehlerIdx := 0;
		bBusy := FALSE;	
	END_IF
END_CASE
END_ACTION

ACTION d_EL1918:

// 16#10F3 ist der Index für den Diag-History-Reiter in der online-Ansicht im EA-Baum
// 16#01: Subindex für das Maximum an Meldungen
// 16#02: Subindex für die neuste Meldung
// 16#03: Subindex für die neuste quittierte Meldung
// 16#04: Subindex eine neue Meldung vorhanden
// 16#05: Subindex für allgemeine Flags
// 16#06 - 16#45: Subindexe für die Meldungen

// Weitere Diagnoseobjekte:
// 16#F984 ist der Index für Device System Data vom Controller 1
// 16#02: Subindex für die Temperatur
// 16#F985 ist der Index für Device System Data vom Controller 2
// 16#02: Subindex für die Temperatur
// Sollten aber auch alle in der Diag History stehen.

// ModuleFault:
// 16#6002:01 Ch1
// 16#6012:01 Ch2
// 16#6022:01 Ch3
// 16#6032:01 Ch4
// 16#6042:01 Ch5
// 16#6052:01 Ch6
// 16#6062:01 Ch7
// 16#6072:01 Ch8

// Eine richtige Diagnose der TwinSAFE-Ein-/ und Ausgänge ist nicht mehr über die CoE-Objekte möglich. Das muss über die DiagHistory gemacht werden. GGf. ist das bald in der HMI
CASE nStateDatenAuslesen OF
	
0:	// EL1918 Diagnose init 
	bBusy 			:= TRUE;	// Solange diese Bit an ist, wird diese Aktion aufgerufen
	nChannelDiag	:= 1;	// Immer bei Kanal 1 beginnen.
	MEMSET(ADR(arrModuleFault),0,SIZEOF(arrModuleFault));	// Rücksetzen
	MEMSET(ADR(arrModuleFaultLink),0,SIZEOF(arrModuleFaultLink));	// Rücksetzen
	
	nStateDatenAuslesen	:= nStateDatenAuslesen +1;
	
1:	// Module Fault der einzelnen Kanäle auslesen: Index errechnen
	
	nCoeIndex		:= 16#6002 + ((nChannelDiag-1)* 16#10);	// Index für ModuleFault pro Kanal
	nCoESubIndex	:= 16#01;	// Index der neusten Meldung
	nStateDatenAuslesen	:= nStateDatenAuslesen +1;
	
2:	// Module Fault der einzelnen Kanäle auslesen: Lesen starten

	fbCoeRead(
		sNetId		:= sEtherCatNetID,
		nSlaveAddr 	:= arrSafetyKlemmeInfo[nAktKlemme].nAdresse,
		nIndex		:= nCoEIndex,
		nSubIndex 	:= nCoESubIndex,
		pDstBuf		:= ADR(nDiagMessage),
		cbBufLen		:= SIZEOF(nDiagMessage),
		bExecute		:= TRUE,

		bError		=> bCoeReadError,
		nErrId		=> nCoeReadErrId
	);
	nStateDatenAuslesen := nStateDatenAuslesen + 1;

3:	// Module Fault der einzelnen Kanäle auslesen: Warten auf gelesen

	fbCoeRead(bExecute:= FALSE);

	IF NOT fbCoeRead.bBusy
	THEN	// Baustein ist durchgelaufen
		IF fbCoeRead.bError
		THEN	// Wenn ein Error vorliegt, wird dieser ausgegeben
			nLastErrIDTemp := fbCoeRead.nErrID;	// Error-ID des CoE Reads wird gespeichert
			bCoeReadError := TRUE;
		ELSE
			bCoeReadError := FALSE;
		END_IF
		
		nStateDatenAuslesen := nStateDatenAuslesen + 1;
	END_IF
	
4:	// Module Fault der einzelnen Kanäle auslesen: Lesen auswerten

	arrModuleFault[nChannelDiag]	:= nDiagMessage <> 0;
	
	IF nChannelDiag = 8
	THEN
		nStateDatenAuslesen := 11;
		nChannelDiag	:= 1;
	ELSE
		nChannelDiag	:= nChannelDiag +1;
		nStateDatenAuslesen := 1;
	END_IF

11:	// Module Fault Link der einzelnen Kanäle auslesen: Index errechnen

// ModuleFaultLink:
// 16#8000:05 Ch1
// 16#8010:05 Ch2
// 16#8020:05 Ch3
// 16#8030:05 Ch4
// 16#8040:05 Ch5
// 16#8050:05 Ch6
// 16#8060:05 Ch7
// 16#8070:05 Ch8

	nCoeIndex		:= 16#8000 + ((nChannelDiag-1)* 16#10);	// Index für ModuleFaultLink pro Kanal
	nCoESubIndex	:= 16#05;	// Index der neusten Meldung
	nStateDatenAuslesen	:= nStateDatenAuslesen +1;
	
12:	// Module Fault Link der einzelnen Kanäle auslesen: Lesen starten

	fbCoeRead(
		sNetId		:= sEtherCatNetID,
		nSlaveAddr 	:= arrSafetyKlemmeInfo[nAktKlemme].nAdresse,
		nIndex		:= nCoEIndex,
		nSubIndex 	:= nCoESubIndex,
		pDstBuf		:= ADR(nDiagMessage),
		cbBufLen		:= SIZEOF(nDiagMessage),
		bExecute		:= TRUE,

		bError		=> bCoeReadError,
		nErrId		=> nCoeReadErrId
	);
	nStateDatenAuslesen := nStateDatenAuslesen + 1;

13:	// Module Fault Link der einzelnen Kanäle auslesen: Warten auf gelesen

	fbCoeRead(bExecute:= FALSE);

	IF NOT fbCoeRead.bBusy
	THEN	// Baustein ist durchgelaufen
		IF fbCoeRead.bError
		THEN	// Wenn ein Error vorliegt, wird dieser ausgegeben
			nLastErrIDTemp := fbCoeRead.nErrID;	// Error-ID des CoE Reads wird gespeichert
			bCoeReadError := TRUE;
		ELSE
			bCoeReadError := FALSE;
		END_IF
		
		nStateDatenAuslesen := nStateDatenAuslesen + 1;
	END_IF
	
14:	// Module Fault Link der einzelnen Kanäle auslesen: Lesen auswerten

	arrModuleFaultLink[nChannelDiag]	:= nDiagMessage <> 0;
	
	IF nChannelDiag = 8
	THEN
		nStateDatenAuslesen := 21;
		nChannelDiag	:= 1;
	ELSE
		nChannelDiag	:= nChannelDiag +1;
		nStateDatenAuslesen := 11;
	END_IF
	
21:	// ModuleFault gesammelt auswerten.

	bModuleFaultActive	:= FALSE;
	FOR nChannelDiag := 1 TO 8 DO
		IF arrModuleFault[nChannelDiag]
		THEN
			bModuleFaultActive	:= TRUE;
		END_IF
	END_FOR
	
	nStateDatenAuslesen := nStateDatenAuslesen + 1;
	
22:	// Fehlermeldung auswerten

	FOR nChannelDiag := 1 TO 8 DO
		IF arrModuleFault[nChannelDiag]
			AND arrModuleFaultLink[nChannelDiag]
		THEN	// Modulfehler mit aktivem ModuleFaultLink
		
			arrSafetyKlemmeInfo[nAktKlemme].arrFehler[nFehlerIdx] := TRUE;
			arrSafetyKlemmeInfo[nAktKlemme].arrFehlertext[nFehlerIdx] := 
				CONCAT('ModuleFault bei Klemme: ',
				CONCAT(arrSafetyKlemmeInfo[nAktKlemme].sName,
				CONCAT(' Kanal: ',
				CONCAT(TO_STRING(nChannelDiag),' Bei aktivem ModuleFaultLink. Der Fehler kann aber auch an einem anderen Kanal liegen.'))));
			nFehlerIdx := nFehlerIdx + 1;
		ELSIF arrModuleFault[nChannelDiag]
		THEN	// Modulfehler ohne ModuleFaultLink. Das heißt, dass der Fehler definitiv an diesem Kanal liegt.
		
			arrSafetyKlemmeInfo[nAktKlemme].arrFehler[nFehlerIdx] := TRUE;
			arrSafetyKlemmeInfo[nAktKlemme].arrFehlertext[nFehlerIdx] := 
				CONCAT('ModuleFault bei Klemme: ',
				CONCAT(arrSafetyKlemmeInfo[nAktKlemme].sName,
				CONCAT(' Kanal: ',TO_STRING(nChannelDiag))));
			nFehlerIdx := nFehlerIdx + 1;
		END_IF
	END_FOR
	
	nStateDatenAuslesen := 99;	// fertig

99:	// Fertig mit auslesen
	
	arrSafetyKlemmeInfo[nAktKlemme].nAnzFehler := nFehlerIdx;
	nStateDatenAuslesen := 0;
	nFehlerIdx := 0; 
	bBusy := FALSE;

END_CASE
END_ACTION

ACTION d_EP1908:
CASE nStateDatenAuslesen OF
0:
	bBusy			:= TRUE;	
	
	nCoeIndex		:= 16#FA80; (*Index fuer die Temperatur*)
	nCoESubIndex	:= 16#1;
	
	(*Auslesen der Temperatur*)
	fbCoeRead(
	sNetId		:= sEtherCatNetID,
	nSlaveAddr 	:= arrSafetyKlemmeInfo[nAktKlemme].nAdresse,
	nIndex		:= nCoEIndex,
	nSubIndex 	:= nCoESubIndex,
	pDstBuf		:= ADR(nReadBuf),
	cbBufLen	:= SIZEOF(nReadBuf),
	bExecute	:= TRUE,

	bError		=> bCoeReadError,
	nErrId		=> nCoeReadErrId
	);
		
	fbCoeRead(bExecute:= FALSE);

	IF NOT fbCoeRead.bBusy THEN					(* Baustein ist durchgelaufen *)
		IF fbCoeRead.bError THEN				(* Wenn ein Error vorliegt, wird dieser ausgegeben *)
			nLastErrIDTemp 
				:= fbCoeRead.nErrID;
			bCoeReadError := TRUE;
		ELSE
			(*Auswertung des Buffers aus dem CoE-Read - Vergleich mit Maximaltemperatur*)
			IF nReadBuf > cMaxTemperatur THEN
				arrSafetyKlemmeInfo[nAktKlemme].arrFehler[nFehlerIdx] := TRUE;
				arrSafetyKlemmeInfo[nAktKlemme].arrFehlertext[nFehlerIdx] := 
					CONCAT('TwinSafe: Maximale Temperatur überschritten an Klemme mit der Adresse: ',
					arrSafetyKlemmeInfo[nAktKlemme].sName);
				nFehlerIdx := nFehlerIdx + 1;
			END_IF
			bCoeReadError := FALSE; 
		END_IF
		nStateDatenAuslesen := nStateDatenAuslesen + 1;	
	END_IF
		
1:
(*Sensortest-Fehler-Überprüfung*)
	nCoeIndex		:= 16#800E; (*Index fuer die Diagnose*)
	nCoESubIndex	:= 16#0A;	(*Sensortest-Fehler-Ueberpruefung*)
	
	(*Auslesen der Diagnose-Informationen*)
	fbCoeRead(
	sNetId		:= sEtherCatNetID,
	nSlaveAddr 	:= arrSafetyKlemmeInfo[nAktKlemme].nAdresse,
	nIndex		:= nCoEIndex,
	nSubIndex 	:= nCoESubIndex,
	pDstBuf		:= ADR(nReadBuf),
	cbBufLen	:= SIZEOF(nReadBuf),
	bExecute	:= TRUE,

	bError		=> bCoeReadError,
	nErrId		=> nCoeReadErrId
	);

	fbCoeRead(bExecute:= FALSE);
	
	IF NOT fbCoeRead.bBusy THEN					(* Baustein ist durchgelaufen *)
		IF fbCoeRead.bError THEN				
			nLastErrIDTemp 
				:= fbCoeRead.nErrID;
			bCoeReadError := TRUE;
		ELSE
			(*Auswertung des Buffers aus dem CoE-Read*)
			IF nReadBuf.0 THEN
				arrSafetyKlemmeInfo[nAktKlemme].arrFehler[nFehlerIdx] := TRUE;
				arrSafetyKlemmeInfo[nAktKlemme].arrFehlertext[nFehlerIdx] := 
					CONCAT('Fehler beim Sensortest der Safety-Klemme! (Adresse: ',
					CONCAT(arrSafetyKlemmeInfo[nAktKlemme].sName,(', Eingang 1)')));
				nFehlerIdx := nFehlerIdx + 1;	
			END_IF
			IF nReadBuf.1 THEN
				arrSafetyKlemmeInfo[nAktKlemme].arrFehler[nFehlerIdx] := TRUE;
				arrSafetyKlemmeInfo[nAktKlemme].arrFehlertext[nFehlerIdx] := 
					CONCAT('Fehler beim Sensortest der Safety-Klemme! (Adresse: ',
					CONCAT(arrSafetyKlemmeInfo[nAktKlemme].sName,(', Eingang 2)')));
				nFehlerIdx := nFehlerIdx + 1;	
			END_IF
			IF nReadBuf.2 THEN
				arrSafetyKlemmeInfo[nAktKlemme].arrFehler[nFehlerIdx] := TRUE;
				arrSafetyKlemmeInfo[nAktKlemme].arrFehlertext[nFehlerIdx] := 
					CONCAT('Fehler beim Sensortest der Safety-Klemme! (Adresse: ',
					CONCAT(arrSafetyKlemmeInfo[nAktKlemme].sName,(', Eingang 3)')));
				nFehlerIdx := nFehlerIdx + 1;
			END_IF	
			IF nReadBuf.3 THEN
				arrSafetyKlemmeInfo[nAktKlemme].arrFehler[nFehlerIdx] := TRUE;
				arrSafetyKlemmeInfo[nAktKlemme].arrFehlertext[nFehlerIdx] := 
					CONCAT('Fehler beim Sensortest der Safety-Klemme! (Adresse: ',
					CONCAT(arrSafetyKlemmeInfo[nAktKlemme].sName,(', Eingang 4)')));
				nFehlerIdx := nFehlerIdx + 1;	
			END_IF
			bCoeReadError := FALSE;
		END_IF
			nStateDatenAuslesen := nStateDatenAuslesen + 1;
	END_IF

2:
	
	nCoeIndex		:= 16#800E; (*Index fuer die Diagnose*)
	nCoESubIndex	:= 16#0B;	(*Fehler bei zweikanaliger Auswertung*)
	
	(*Auslesen der Diagnose-Informationen*)
	fbCoeRead(
	sNetId		:= sEtherCatNetID,
	nSlaveAddr 	:= arrSafetyKlemmeInfo[nAktKlemme].nAdresse,
	nIndex		:= nCoEIndex,
	nSubIndex 	:= nCoESubIndex,
	pDstBuf		:= ADR(nReadBuf),
	cbBufLen	:= SIZEOF(nReadBuf),
	bExecute	:= TRUE,

	bError		=> bCoeReadError,
	nErrId		=> nCoeReadErrId
	);

	fbCoeRead(bExecute:= FALSE);
	
	IF NOT fbCoeRead.bBusy THEN					(* Baustein ist durchgelaufen *)
		IF fbCoeRead.bError THEN				(* Wenn ein Error vorliegt, wird dieser ausgegeben *)
			nLastErrIDTemp 
				:= fbCoeRead.nErrID;
			bCoeReadError := TRUE;
		ELSE
			(*Auswertung des Buffers aus dem CoE-Read*)
			IF nReadBuf.0 THEN
				arrSafetyKlemmeInfo[nAktKlemme].arrFehler[nFehlerIdx] := TRUE;
				arrSafetyKlemmeInfo[nAktKlemme].arrFehlertext[nFehlerIdx] := 
					CONCAT('TwinSAFE: Fehler bei zweikanaliger Auswertung an Adresse:',
					arrSafetyKlemmeInfo[nAktKlemme].sName);
				nFehlerIdx := nFehlerIdx + 1;
			END_IF
			bCoeReadError := FALSE;
		END_IF
			nStateDatenAuslesen := nStateDatenAuslesen + 1;
	END_IF

3:
	nCoeIndex		:= 16#800E; (*Index fuer die Diagnose*)
	nCoESubIndex	:= 16#0C;	(*Fehler bei Trittmattenbetriebsart: Eingangspaar uneinig*)
	
	(*Auslesen der Diagnose-Informationen*)
	fbCoeRead(
	sNetId		:= sEtherCatNetID,
	nSlaveAddr 	:= arrSafetyKlemmeInfo[nAktKlemme].nAdresse,
	nIndex		:= nCoEIndex,
	nSubIndex 	:= nCoESubIndex,
	pDstBuf		:= ADR(nReadBuf),
	cbBufLen	:= SIZEOF(nReadBuf),
	bExecute	:= TRUE,

	bError		=> bCoeReadError,
	nErrId		=> nCoeReadErrId
	);

	fbCoeRead(bExecute:= FALSE);
	IF NOT fbCoeRead.bBusy THEN				(* Baustein ist durchgelaufen *)
		IF fbCoeRead.bError THEN				(* Wenn ein Error vorliegt, wird dieser ausgegeben *)
			nLastErrIDTemp 
				:= fbCoeRead.nErrID;
			bCoeReadError := TRUE;
		ELSE
			(*Auswertung des Buffers aus dem CoE-Read*)
			IF nReadBuf.0 THEN
				arrSafetyKlemmeInfo[nAktKlemme].arrFehler[nFehlerIdx] := TRUE;
				arrSafetyKlemmeInfo[nAktKlemme].arrFehlertext[nFehlerIdx] := 
					CONCAT('TwinSAFE: Fehler bei Trittmattenbetriebsart (Eingangspaar uneinig) an Adresse:',
					arrSafetyKlemmeInfo[nAktKlemme].sName);
				nFehlerIdx := nFehlerIdx + 1;
			END_IF
			bCoeReadError := FALSE;
		END_IF
			nStateDatenAuslesen := nStateDatenAuslesen + 1;
	END_IF

4:	
	nCoeIndex		:= 16#800E; (*Index fuer die Diagnose*)
	nCoESubIndex	:= 16#0D;	(*Fehler bei Trittmattenbetriebsart: Fremdeinspeisung*)
	
	(*Auslesen der Diagnose-Informationen*)
	fbCoeRead(
	sNetId		:= sEtherCatNetID,
	nSlaveAddr 	:= arrSafetyKlemmeInfo[nAktKlemme].nAdresse,
	nIndex		:= nCoEIndex,
	nSubIndex 	:= nCoESubIndex,
	pDstBuf		:= ADR(nReadBuf),
	cbBufLen	:= SIZEOF(nReadBuf),
	bExecute	:= TRUE,

	bError		=> bCoeReadError,
	nErrId		=> nCoeReadErrId
	);

	fbCoeRead(bExecute:= FALSE);
	IF NOT fbCoeRead.bBusy THEN					(* Baustein ist durchgelaufen *)
		IF fbCoeRead.bError THEN				(* Wenn ein Error vorliegt, wird dieser ausgegeben *)
			nLastErrIDTemp 
				:= fbCoeRead.nErrID;
			bCoeReadError := TRUE;
		ELSE
			(*Auswertung des Buffers aus dem CoE-Read*)
			IF nReadBuf.0 THEN
				arrSafetyKlemmeInfo[nAktKlemme].arrFehler[nFehlerIdx] := TRUE;
				arrSafetyKlemmeInfo[nAktKlemme].arrFehlertext[nFehlerIdx] := 
					CONCAT('TwinSAFE: Fehler bei Trittmattenbetriebsart (Fremdeinspeisung) an Adresse:',
					arrSafetyKlemmeInfo[nAktKlemme].sName);
				nFehlerIdx := nFehlerIdx + 1;
			END_IF
			bCoeReadError := FALSE;
		END_IF
		nStateDatenAuslesen := 0;	
		arrSafetyKlemmeInfo[nAktKlemme].nAnzFehler := nFehlerIdx;
		nFehlerIdx := 0;
		bBusy := FALSE;	
	END_IF
END_CASE
END_ACTION

ACTION d_EP1918:

// 16#10F3 ist der Index für den Diag-History-Reiter in der online-Ansicht im EA-Baum
// 16#01: Subindex für das Maximum an Meldungen
// 16#02: Subindex für die neuste Meldung
// 16#03: Subindex für die neuste quittierte Meldung
// 16#04: Subindex eine neue Meldung vorhanden
// 16#05: Subindex für allgemeine Flags
// 16#06 - 16#45: Subindexe für die Meldungen

// Weitere Diagnoseobjekte:
// 16#F984 ist der Index für Device System Data vom Controller 1
// 16#02: Subindex für die Temperatur
// 16#F985 ist der Index für Device System Data vom Controller 2
// 16#02: Subindex für die Temperatur
// Sollten aber auch alle in der Diag History stehen.

// ModuleFault:
// 16#6002:01 Ch1
// 16#6012:01 Ch2
// 16#6022:01 Ch3
// 16#6032:01 Ch4
// 16#6042:01 Ch5
// 16#6052:01 Ch6
// 16#6062:01 Ch7
// 16#6072:01 Ch8

// Eine richtige Diagnose der TwinSAFE-Ein-/ und Ausgänge ist nicht mehr über die CoE-Objekte möglich. Das muss über die DiagHistory gemacht werden. GGf. ist das bald in der HMI
CASE nStateDatenAuslesen OF
	
0:	// EL1918 Diagnose init 
	bBusy 			:= TRUE;	// Solange diese Bit an ist, wird diese Aktion aufgerufen
	nChannelDiag	:= 1;	// Immer bei Kanal 1 beginnen.
	MEMSET(ADR(arrModuleFault),0,SIZEOF(arrModuleFault));	// Rücksetzen
	MEMSET(ADR(arrModuleFaultLink),0,SIZEOF(arrModuleFaultLink));	// Rücksetzen
	
	nStateDatenAuslesen	:= nStateDatenAuslesen +1;
	
1:	// Module Fault der einzelnen Kanäle auslesen: Index errechnen
	
	nCoeIndex		:= 16#6002 + ((nChannelDiag-1)* 16#10);	// Index für ModuleFault pro Kanal
	nCoESubIndex	:= 16#01;	// Index der neusten Meldung
	nStateDatenAuslesen	:= nStateDatenAuslesen +1;
	
2:	// Module Fault der einzelnen Kanäle auslesen: Lesen starten

	fbCoeRead(
		sNetId		:= sEtherCatNetID,
		nSlaveAddr 	:= arrSafetyKlemmeInfo[nAktKlemme].nAdresse,
		nIndex		:= nCoEIndex,
		nSubIndex 	:= nCoESubIndex,
		pDstBuf		:= ADR(nDiagMessage),
		cbBufLen		:= SIZEOF(nDiagMessage),
		bExecute		:= TRUE,

		bError		=> bCoeReadError,
		nErrId		=> nCoeReadErrId
	);
	nStateDatenAuslesen := nStateDatenAuslesen + 1;

3:	// Module Fault der einzelnen Kanäle auslesen: Warten auf gelesen

	fbCoeRead(bExecute:= FALSE);

	IF NOT fbCoeRead.bBusy
	THEN	// Baustein ist durchgelaufen
		IF fbCoeRead.bError
		THEN	// Wenn ein Error vorliegt, wird dieser ausgegeben
			nLastErrIDTemp := fbCoeRead.nErrID;	// Error-ID des CoE Reads wird gespeichert
			bCoeReadError := TRUE;
		ELSE
			bCoeReadError := FALSE;
		END_IF
		
		nStateDatenAuslesen := nStateDatenAuslesen + 1;
	END_IF
	
4:	// Module Fault der einzelnen Kanäle auslesen: Lesen auswerten

	arrModuleFault[nChannelDiag]	:= nDiagMessage <> 0;
	
	IF nChannelDiag = 8
	THEN
		nStateDatenAuslesen := 11;
		nChannelDiag	:= 1;
	ELSE
		nChannelDiag	:= nChannelDiag +1;
		nStateDatenAuslesen := 1;
	END_IF

11:	// Module Fault Link der einzelnen Kanäle auslesen: Index errechnen

// ModuleFaultLink:
// 16#8000:05 Ch1
// 16#8010:05 Ch2
// 16#8020:05 Ch3
// 16#8030:05 Ch4
// 16#8040:05 Ch5
// 16#8050:05 Ch6
// 16#8060:05 Ch7
// 16#8070:05 Ch8

	nCoeIndex		:= 16#8000 + ((nChannelDiag-1)* 16#10);	// Index für ModuleFaultLink pro Kanal
	nCoESubIndex	:= 16#05;	// Index der neusten Meldung
	nStateDatenAuslesen	:= nStateDatenAuslesen +1;
	
12:	// Module Fault Link der einzelnen Kanäle auslesen: Lesen starten

	fbCoeRead(
		sNetId		:= sEtherCatNetID,
		nSlaveAddr 	:= arrSafetyKlemmeInfo[nAktKlemme].nAdresse,
		nIndex		:= nCoEIndex,
		nSubIndex 	:= nCoESubIndex,
		pDstBuf		:= ADR(nDiagMessage),
		cbBufLen		:= SIZEOF(nDiagMessage),
		bExecute		:= TRUE,

		bError		=> bCoeReadError,
		nErrId		=> nCoeReadErrId
	);
	nStateDatenAuslesen := nStateDatenAuslesen + 1;

13:	// Module Fault Link der einzelnen Kanäle auslesen: Warten auf gelesen

	fbCoeRead(bExecute:= FALSE);

	IF NOT fbCoeRead.bBusy
	THEN	// Baustein ist durchgelaufen
		IF fbCoeRead.bError
		THEN	// Wenn ein Error vorliegt, wird dieser ausgegeben
			nLastErrIDTemp := fbCoeRead.nErrID;	// Error-ID des CoE Reads wird gespeichert
			bCoeReadError := TRUE;
		ELSE
			bCoeReadError := FALSE;
		END_IF
		
		nStateDatenAuslesen := nStateDatenAuslesen + 1;
	END_IF
	
14:	// Module Fault Link der einzelnen Kanäle auslesen: Lesen auswerten

	arrModuleFaultLink[nChannelDiag]	:= nDiagMessage <> 0;
	
	IF nChannelDiag = 8
	THEN
		nStateDatenAuslesen := 21;
		nChannelDiag	:= 1;
	ELSE
		nChannelDiag	:= nChannelDiag +1;
		nStateDatenAuslesen := 11;
	END_IF
	
21:	// ModuleFault gesammelt auswerten.

	bModuleFaultActive	:= FALSE;
	FOR nChannelDiag := 1 TO 8 DO
		IF arrModuleFault[nChannelDiag]
		THEN
			bModuleFaultActive	:= TRUE;
		END_IF
	END_FOR
	
	nStateDatenAuslesen := nStateDatenAuslesen + 1;
	
22:	// Fehlermeldung auswerten

	FOR nChannelDiag := 1 TO 8 DO
		IF arrModuleFault[nChannelDiag]
			AND arrModuleFaultLink[nChannelDiag]
		THEN	// Modulfehler mit aktivem ModuleFaultLink
		
			arrSafetyKlemmeInfo[nAktKlemme].arrFehler[nFehlerIdx] := TRUE;
			arrSafetyKlemmeInfo[nAktKlemme].arrFehlertext[nFehlerIdx] := 
				CONCAT('ModuleFault bei Klemme: ',
				CONCAT(arrSafetyKlemmeInfo[nAktKlemme].sName,
				CONCAT(' Kanal: ',
				CONCAT(TO_STRING(nChannelDiag),' Bei aktivem ModuleFaultLink. Der Fehler kann aber auch an einem anderen Kanal liegen.'))));
			nFehlerIdx := nFehlerIdx + 1;
		ELSIF arrModuleFault[nChannelDiag]
		THEN	// Modulfehler ohne ModuleFaultLink. Das heißt, dass der Fehler definitiv an diesem Kanal liegt.
		
			arrSafetyKlemmeInfo[nAktKlemme].arrFehler[nFehlerIdx] := TRUE;
			arrSafetyKlemmeInfo[nAktKlemme].arrFehlertext[nFehlerIdx] := 
				CONCAT('ModuleFault bei Klemme: ',
				CONCAT(arrSafetyKlemmeInfo[nAktKlemme].sName,
				CONCAT(' Kanal: ',TO_STRING(nChannelDiag))));
			nFehlerIdx := nFehlerIdx + 1;
		END_IF
	END_FOR
	
	nStateDatenAuslesen := 99;	// fertig

99:	// Fertig mit auslesen
	
	arrSafetyKlemmeInfo[nAktKlemme].nAnzFehler := nFehlerIdx;
	nStateDatenAuslesen := 0;
	nFehlerIdx := 0; 
	bBusy := FALSE;

END_CASE
END_ACTION

ACTION d_EP1957:
// Safety-EP-Box mit 4 Eingänge und 4 Ausgänge

// Weitere Diagnoseobjekte:
// 16#F984 ist der Index für Device System Data vom Controller 1
// 16#02: Subindex für die Temperatur
// 16#F985 ist der Index für Device System Data vom Controller 2
// 16#02: Subindex für die Temperatur
// Sollten aber auch alle in der Diag History stehen.

// ModuleFault:
// 16#6002:01 Ch1 Out
// 16#6012:01 Ch2 Out
// 16#6022:01 Ch3 Out
// 16#6032:01 Ch4 Out
// 16#6042:01 Ch1 In
// 16#6052:01 Ch2 In
// 16#6062:01 Ch3 In
// 16#6072:01 Ch4 In

// Eine richtige Diagnose der TwinSAFE-Ein-/ und Ausgänge ist nicht mehr über die CoE-Objekte möglich. Das muss über die DiagHistory gemacht werden. GGf. ist das bald in der HMI
CASE nStateDatenAuslesen OF
	
0:	// EL1957 Diagnose init 
	bBusy 			:= TRUE;	// Solange diese Bit an ist, wird diese Aktion aufgerufen
	nChannelDiag	:= 1;	// Immer bei Kanal 1 beginnen.
	MEMSET(ADR(arrModuleFault),0,SIZEOF(arrModuleFault));	// Rücksetzen
	MEMSET(ADR(arrModuleFaultLink),0,SIZEOF(arrModuleFaultLink));	// Rücksetzen
	
	nStateDatenAuslesen	:= nStateDatenAuslesen +1;
	
1:	// Module Fault der einzelnen Kanäle auslesen: Index errechnen
	
	nCoeIndex		:= 16#6002 + ((nChannelDiag-1)* 16#10);	// Index für ModuleFault pro Kanal
	nCoESubIndex	:= 16#01;
	nStateDatenAuslesen	:= nStateDatenAuslesen +1;
	
2:	// Module Fault der einzelnen Kanäle auslesen: Lesen starten

	fbCoeRead(
		sNetId		:= sEtherCatNetID,
		nSlaveAddr 	:= arrSafetyKlemmeInfo[nAktKlemme].nAdresse,
		nIndex		:= nCoEIndex,
		nSubIndex 	:= nCoESubIndex,
		pDstBuf		:= ADR(nDiagMessage),
		cbBufLen		:= SIZEOF(nDiagMessage),
		bExecute		:= TRUE,

		bError		=> bCoeReadError,
		nErrId		=> nCoeReadErrId
	);
	nStateDatenAuslesen := nStateDatenAuslesen + 1;

3:	// Module Fault der einzelnen Kanäle auslesen: Warten auf gelesen

	fbCoeRead(bExecute:= FALSE);

	IF NOT fbCoeRead.bBusy
	THEN	// Baustein ist durchgelaufen
		IF fbCoeRead.bError
		THEN	// Wenn ein Error vorliegt, wird dieser ausgegeben
			nLastErrIDTemp := fbCoeRead.nErrID;	// Error-ID des CoE Reads wird gespeichert
			bCoeReadError := TRUE;
		ELSE
			bCoeReadError := FALSE;
		END_IF
		
		nStateDatenAuslesen := nStateDatenAuslesen + 1;
	END_IF
	
4:	// Module Fault der einzelnen Kanäle auslesen: Lesen auswerten

	arrModuleFault[nChannelDiag]	:= nDiagMessage <> 0;
	
	IF nChannelDiag = 8
	THEN
		nStateDatenAuslesen := 11;
		nChannelDiag	:= 1;
	ELSE
		nChannelDiag	:= nChannelDiag +1;
		nStateDatenAuslesen := 1;
	END_IF

11:	// Module Fault Link der einzelnen Kanäle auslesen: Index errechnen

// ModuleFaultLink:
// 16#8000:07 Ch1 Out
// 16#8010:07 Ch2 Out
// 16#8020:07 Ch3 Out
// 16#8030:07 Ch4 Out
// 16#8040:05 Ch1 In 
// 16#8050:05 Ch2 In 
// 16#8060:05 Ch3 In 
// 16#8070:05 Ch4 In 

	nCoeIndex		:= 16#8000 + ((nChannelDiag-1)* 16#10);	// Index für ModuleFaultLink pro Kanal
	
	IF nChannelDiag > 4
	THEN
		nCoESubIndex	:= 16#07;	// Sub-Index für Ausgänge
	ELSE
		nCoESubIndex	:= 16#05;	// Sub-Index für Eingänge
	END_IF
	
	nStateDatenAuslesen	:= nStateDatenAuslesen +1;
	
12:	// Module Fault Link der einzelnen Kanäle auslesen: Lesen starten

	fbCoeRead(
		sNetId		:= sEtherCatNetID,
		nSlaveAddr 	:= arrSafetyKlemmeInfo[nAktKlemme].nAdresse,
		nIndex		:= nCoEIndex,
		nSubIndex 	:= nCoESubIndex,
		pDstBuf		:= ADR(nDiagMessage),
		cbBufLen		:= SIZEOF(nDiagMessage),
		bExecute		:= TRUE,

		bError		=> bCoeReadError,
		nErrId		=> nCoeReadErrId
	);
	nStateDatenAuslesen := nStateDatenAuslesen + 1;

13:	// Module Fault Link der einzelnen Kanäle auslesen: Warten auf gelesen

	fbCoeRead(bExecute:= FALSE);

	IF NOT fbCoeRead.bBusy
	THEN	// Baustein ist durchgelaufen
		IF fbCoeRead.bError
		THEN	// Wenn ein Error vorliegt, wird dieser ausgegeben
			nLastErrIDTemp := fbCoeRead.nErrID;	// Error-ID des CoE Reads wird gespeichert
			bCoeReadError := TRUE;
		ELSE
			bCoeReadError := FALSE;
		END_IF
		
		nStateDatenAuslesen := nStateDatenAuslesen + 1;
	END_IF
	
14:	// Module Fault Link der einzelnen Kanäle auslesen: Lesen auswerten

	arrModuleFaultLink[nChannelDiag]	:= nDiagMessage <> 0;
	
	IF nChannelDiag = 8
	THEN
		nStateDatenAuslesen := 21;
		nChannelDiag	:= 1;
	ELSE
		nChannelDiag	:= nChannelDiag +1;
		nStateDatenAuslesen := 11;
	END_IF
	
21:	// ModuleFault gesammelt auswerten.

	bModuleFaultActive	:= FALSE;
	FOR nChannelDiag := 1 TO 8 DO
		IF arrModuleFault[nChannelDiag]
		THEN
			bModuleFaultActive	:= TRUE;
		END_IF
	END_FOR
	
	nStateDatenAuslesen := nStateDatenAuslesen + 1;
	
22:	// Fehlermeldung auswerten

	FOR nChannelDiag := 1 TO 8 DO
		IF arrModuleFault[nChannelDiag]
			AND arrModuleFaultLink[nChannelDiag]
		THEN	// Modulfehler mit aktivem ModuleFaultLink
			IF nChannelDiag > 4
			THEN
				arrSafetyKlemmeInfo[nAktKlemme].arrFehler[nFehlerIdx] := TRUE;
				arrSafetyKlemmeInfo[nAktKlemme].arrFehlertext[nFehlerIdx] := 
					CONCAT('ModuleFault bei Klemme: ',
					CONCAT(arrSafetyKlemmeInfo[nAktKlemme].sName,
					CONCAT(' Eingangs-Kanal: ',
					CONCAT(TO_STRING(nChannelDiag-4),' Bei aktivem ModuleFaultLink. Der Fehler kann aber auch an einem anderen Kanal liegen.'))));
				nFehlerIdx := nFehlerIdx + 1;
			ELSE
				arrSafetyKlemmeInfo[nAktKlemme].arrFehler[nFehlerIdx] := TRUE;
				arrSafetyKlemmeInfo[nAktKlemme].arrFehlertext[nFehlerIdx] := 
					CONCAT('ModuleFault bei Klemme: ',
					CONCAT(arrSafetyKlemmeInfo[nAktKlemme].sName,
					CONCAT(' Ausgangs-Kanal: ',
					CONCAT(TO_STRING(nChannelDiag),' Bei aktivem ModuleFaultLink. Der Fehler kann aber auch an einem anderen Kanal liegen.'))));
				nFehlerIdx := nFehlerIdx + 1;
			END_IF
		ELSIF arrModuleFault[nChannelDiag]
		THEN	// Modulfehler ohne ModuleFaultLink. Das heißt, dass der Fehler definitiv an diesem Kanal liegt.
			IF nChannelDiag > 4
			THEN
				arrSafetyKlemmeInfo[nAktKlemme].arrFehler[nFehlerIdx] := TRUE;
				arrSafetyKlemmeInfo[nAktKlemme].arrFehlertext[nFehlerIdx] := 
					CONCAT('ModuleFault bei Klemme: ',
					CONCAT(arrSafetyKlemmeInfo[nAktKlemme].sName,
					CONCAT(' Eingangs-Kanal: ',TO_STRING(nChannelDiag-4))));
				nFehlerIdx := nFehlerIdx + 1;
			ELSE
				arrSafetyKlemmeInfo[nAktKlemme].arrFehler[nFehlerIdx] := TRUE;
				arrSafetyKlemmeInfo[nAktKlemme].arrFehlertext[nFehlerIdx] := 
					CONCAT('ModuleFault bei Klemme: ',
					CONCAT(arrSafetyKlemmeInfo[nAktKlemme].sName,
					CONCAT(' Ausgangs-Kanal: ',TO_STRING(nChannelDiag))));
				nFehlerIdx := nFehlerIdx + 1;
			END_IF
		END_IF
	END_FOR
	
	nStateDatenAuslesen := 99;	// Fertig
	
99:	// Fertig mit auslesen
	
	arrSafetyKlemmeInfo[nAktKlemme].nAnzFehler := nFehlerIdx;
	nStateDatenAuslesen := 0;
	nFehlerIdx := 0; 
	bBusy := FALSE;

END_CASE
END_ACTION

ACTION e_EL2904:
CASE nStateDatenAuslesen OF
0:
	bBusy			:= TRUE;	
	
	nCoeIndex		:= 16#FA80; (*Index fuer die Temperatur*)
	nCoESubIndex	:= 16#1;
	
	(*Auslesen der Temperatur*)
	fbCoeRead(
	sNetId		:= sEtherCatNetID,
	nSlaveAddr 	:= arrSafetyKlemmeInfo[nAktKlemme].nAdresse,
	nIndex		:= nCoEIndex,
	nSubIndex 	:= nCoESubIndex,
	pDstBuf		:= ADR(nReadBuf),
	cbBufLen	:= SIZEOF(nReadBuf),
	bExecute	:= TRUE,

	bError		=> bCoeReadError,
	nErrId		=> nCoeReadErrId
	);
		
	fbCoeRead(bExecute:= FALSE);

		IF NOT fbCoeRead.bBusy THEN				(* Baustein ist durchgelaufen *)
			IF fbCoeRead.bError THEN				(* Wenn ein Error vorliegt, wird dieser ausgegeben *)
				nLastErrIDTemp 
					:= fbCoeRead.nErrID;
				bCoeReadError := TRUE;
			ELSE
				bCoeReadError := FALSE;
				(*Abfrage, ob Maximaltemperatur überschritten wird - wenn ja, entsprechendes Bit setzen*)
				IF NOT fbCoeRead.bError 
					AND nReadBuf > cMaxTemperatur THEN
						arrSafetyKlemmeInfo[nAktKlemme].arrFehler[nFehlerIdx] := TRUE;
						arrSafetyKlemmeInfo[nAktKlemme].arrFehlertext[nFehlerIdx] := 
							CONCAT('TwinSafe: Maximale Temperatur überschritten an Klemme mit der Adresse: ',
							arrSafetyKlemmeInfo[nAktKlemme].sName);
						nFehlerIdx := nFehlerIdx + 1;
				ELSIF NOT fbCoeRead.bError THEN
						arrSafetyKlemmeInfo[nAktKlemme].arrFehler[nFehlerIdx] := FALSE;
						arrSafetyKlemmeInfo[nAktKlemme].arrFehlertext[nFehlerIdx] := '';
				END_IF
			END_IF
			nStateDatenAuslesen := nStateDatenAuslesen + 1;	
		END_IF
		
1:
(*Sensortest-Fehler-Überprüfung*)
	nCoeIndex		:= 16#800E; (*Index fuer die Diagnose*)
	nCoESubIndex	:= 16#0C;	(*Sensortest-Fehler-Ueberpruefung*)
	
	(*Auslesen der Diagnose-Informationen*)
	fbCoeRead(
	sNetId		:= sEtherCatNetID,
	nSlaveAddr 	:= arrSafetyKlemmeInfo[nAktKlemme].nAdresse,
	nIndex		:= nCoEIndex,
	nSubIndex 	:= nCoESubIndex,
	pDstBuf		:= ADR(nReadBuf),
	cbBufLen	:= SIZEOF(nReadBuf),
	bExecute	:= TRUE,

	bError		=> bCoeReadError,
	nErrId		=> nCoeReadErrId
	);

	fbCoeRead(bExecute:= FALSE);
	IF NOT fbCoeRead.bBusy THEN					(* Baustein ist durchgelaufen *)
		IF fbCoeRead.bError THEN				(* Wenn ein Error vorliegt, wird dieser ausgegeben; 0 = kein Fehler, 1= Eingang 1; 2= Eingang 2; 3= Eingang 3; 4 = Eingang 4*)
			nLastErrIDTemp 
				:= fbCoeRead.nErrID;
			bCoeReadError := TRUE;
		ELSE
			(*Fehler am Ausgang - Fremdeinspeisung oder Querschluss*)
			IF nReadBuf.0 THEN
				arrSafetyKlemmeInfo[nAktKlemme].arrFehler[nFehlerIdx] := TRUE;
				arrSafetyKlemmeInfo[nAktKlemme].arrFehlertext[nFehlerIdx] := 
					CONCAT('Fehler an Ausgang 1 der Safety-Klemme! Ausgang auf Fremdeinspeisung und Querschluss prüfen! Adresse: ',
						arrSafetyKlemmeInfo[nAktKlemme].sName);
				nFehlerIdx := nFehlerIdx + 1;
			END_IF	
			IF nReadBuf.1 THEN
				arrSafetyKlemmeInfo[nAktKlemme].arrFehler[nFehlerIdx] := TRUE;
				arrSafetyKlemmeInfo[nAktKlemme].arrFehlertext[nFehlerIdx] := 
					CONCAT('Fehler an Ausgang 2 der Safety-Klemme! Ausgang auf Fremdeinspeisung und Querschluss prüfen! Adresse: ',
						arrSafetyKlemmeInfo[nAktKlemme].sName);
				nFehlerIdx := nFehlerIdx + 1;	
			END_IF	
			IF  nReadBuf.2 THEN
				arrSafetyKlemmeInfo[nAktKlemme].arrFehler[nFehlerIdx] := TRUE;
				arrSafetyKlemmeInfo[nAktKlemme].arrFehlertext[nFehlerIdx] := 
					CONCAT('Fehler an Ausgang 3 der Safety-Klemme! Ausgang auf Fremdeinspeisung und Querschluss prüfen! Adresse: ',
						arrSafetyKlemmeInfo[nAktKlemme].sName);
				nFehlerIdx := nFehlerIdx + 1;	
			END_IF	
			IF nReadBuf.3 THEN
				arrSafetyKlemmeInfo[nAktKlemme].arrFehler[nFehlerIdx] := TRUE;
				arrSafetyKlemmeInfo[nAktKlemme].arrFehlertext[nFehlerIdx] := 
					CONCAT('Fehler an Ausgang 4 der Safety-Klemme! Ausgang auf Fremdeinspeisung und Querschluss prüfen! Adresse: ',
						UDINT_TO_STRING(nSlaveAddr));
				nFehlerIdx := nFehlerIdx + 1;	
			END_IF
			(*Fehler am Ausgang - Open Load oder Mindeststrom unterschritten / Höchststrom überschritten*)
			IF nReadBuf.4 THEN
				arrSafetyKlemmeInfo[nAktKlemme].arrFehler[nFehlerIdx] := TRUE;
				arrSafetyKlemmeInfo[nAktKlemme].arrFehlertext[nFehlerIdx] := 
					CONCAT('Fehler an Ausgang 1 der Safety-Klemme! Ausgang im Leerlauf oder Mindeststrom unterschritten / Hoechststrom ueberschritten! Adresse: ',
						arrSafetyKlemmeInfo[nAktKlemme].sName);
				nFehlerIdx := nFehlerIdx + 1;	
			END_IF
			IF nReadBuf.5 THEN
				arrSafetyKlemmeInfo[nAktKlemme].arrFehler[nFehlerIdx] := TRUE;
				arrSafetyKlemmeInfo[nAktKlemme].arrFehlertext[nFehlerIdx] := 
					CONCAT('Fehler an Ausgang 4 der Safety-Klemme! Klemme auf Fremdeinspeisung und Querschluss prüfen! Adresse: ',
						arrSafetyKlemmeInfo[nAktKlemme].sName);
				nFehlerIdx := nFehlerIdx + 1;	
			END_IF	
			IF nReadBuf.6 THEN
				arrSafetyKlemmeInfo[nAktKlemme].arrFehler[nFehlerIdx] := TRUE;
				arrSafetyKlemmeInfo[nAktKlemme].arrFehlertext[nFehlerIdx] := 
					CONCAT('Fehler an Ausgang 4 der Safety-Klemme! Klemme auf Fremdeinspeisung und Querschluss prüfen! Adresse: ',
						arrSafetyKlemmeInfo[nAktKlemme].sName);
				nFehlerIdx := nFehlerIdx + 1;	
			END_IF	
			IF nReadBuf.7 THEN
				arrSafetyKlemmeInfo[nAktKlemme].arrFehler[nFehlerIdx] := TRUE;
				arrSafetyKlemmeInfo[nAktKlemme].arrFehlertext[nFehlerIdx] := 
					CONCAT('Fehler an Ausgang 4 der Safety-Klemme! Klemme auf Fremdeinspeisung und Querschluss prüfen! Adresse: ',
						arrSafetyKlemmeInfo[nAktKlemme].sName);
				nFehlerIdx := nFehlerIdx + 1;	
			END_IF	
			bCoeReadError := FALSE;
		END_IF
			nStateDatenAuslesen := nStateDatenAuslesen + 1;
	END_IF

2:
	
	nCoeIndex		:= 16#800E; (*Index fuer die Diagnose*)
	nCoESubIndex	:= 16#0D;	(*Fehler bei zweikanaliger Auswertung*)
	
	(*Auslesen der Diagnose-Informationen*)
	fbCoeRead(
	sNetId		:= sEtherCatNetID,
	nSlaveAddr 	:= arrSafetyKlemmeInfo[nAktKlemme].nAdresse,
	nIndex		:= nCoEIndex,
	nSubIndex 	:= nCoESubIndex,
	pDstBuf		:= ADR(nReadBuf),
	cbBufLen	:= SIZEOF(nReadBuf),
	bExecute	:= TRUE,

	bError		=> bCoeReadError,
	nErrId		=> nCoeReadErrId
	);

	fbCoeRead(bExecute:= FALSE);
	IF NOT fbCoeRead.bBusy THEN					(* Baustein ist durchgelaufen *)
		IF fbCoeRead.bError THEN				(* Wenn ein Error vorliegt, wird dieser ausgegeben *)
			nLastErrIDTemp 
				:= fbCoeRead.nErrID;
			bCoeReadError := TRUE;
		ELSE
			(*Fehler am Ausgang - Fremdeinspeisung oder Querschluss*)
			IF nReadBuf.0 THEN
				arrSafetyKlemmeInfo[nAktKlemme].arrFehler[nFehlerIdx] := TRUE;
				arrSafetyKlemmeInfo[nAktKlemme].arrFehlertext[nFehlerIdx] := 
					CONCAT('Fehler an Safety-Klemme! Feldspannung zu hoch! Adresse: ',
						arrSafetyKlemmeInfo[nAktKlemme].sName);
				nFehlerIdx := nFehlerIdx + 1;
			END_IF	
			IF nReadBuf.1 THEN
				arrSafetyKlemmeInfo[nAktKlemme].arrFehler[nFehlerIdx] := TRUE;
				arrSafetyKlemmeInfo[nAktKlemme].arrFehlertext[nFehlerIdx] := 
					CONCAT('Fehler an Safety-Klemme! Feldspannung zu niedrig! Adresse: ',
						arrSafetyKlemmeInfo[nAktKlemme].sName);
				nFehlerIdx := nFehlerIdx + 1;	
			END_IF	
			bCoeReadError := FALSE;
		END_IF
			nStateDatenAuslesen := nStateDatenAuslesen + 1;
	END_IF

3:
	nCoeIndex		:= 16#800E; (*Index fuer die Diagnose*)
	nCoESubIndex	:= 16#0E;	(*Klemmentemperaturfehler*)
	
	(*Auslesen der Diagnose-Informationen*)
	fbCoeRead(
	sNetId		:= sEtherCatNetID,
	nSlaveAddr 	:= arrSafetyKlemmeInfo[nAktKlemme].nAdresse,
	nIndex		:= nCoEIndex,
	nSubIndex 	:= nCoESubIndex,
	pDstBuf		:= ADR(nReadBuf),
	cbBufLen	:= SIZEOF(nReadBuf),
	bExecute	:= TRUE,

	bError		=> bCoeReadError,
	nErrId		=> nCoeReadErrId
	);

